  PROC DrawPart48()
    MoveL Offs(pOrigin,340.15,243.37,0.00),v40,z0,tPen\WObj:=wPaper;
    MoveL Offs(pOrigin,341.95,245.18,0.00),v40,z0,tPen\WObj:=wPaper;
    MoveL Offs(pOrigin,341.67,245.49,0.00),v40,z0,tPen\WObj:=wPaper;
    MoveL Offs(pOrigin,344.68,242.48,0.00),v40,z0,tPen\WObj:=wPaper;
    MoveL Offs(pOrigin,344.35,243.09,0.00),v40,z0,tPen\WObj:=wPaper;
    MoveL Offs(pOrigin,346.00,244.74,0.00),v40,z0,tPen\WObj:=wPaper;
    MoveL Offs(pOrigin,346.47,245.17,0.00),v40,z0,tPen\WObj:=wPaper;
    MoveL Offs(pOrigin,349.92,241.72,0.00),v40,z0,tPen\WObj:=wPaper;
    MoveL Offs(pOrigin,349.89,242.65,0.00),v40,z0,tPen\WObj:=wPaper;
    MoveL Offs(pOrigin,351.54,244.31,0.00),v40,z0,tPen\WObj:=wPaper;
    MoveL Offs(pOrigin,351.41,244.71,0.00),v40,z0,tPen\WObj:=wPaper;
    MoveL Offs(pOrigin,354.87,241.25,0.00),v40,z0,tPen\WObj:=wPaper;
    MoveL Offs(pOrigin,355.13,241.92,0.00),v40,z0,tPen\WObj:=wPaper;
    MoveL Offs(pOrigin,356.93,243.72,0.00),v40,z0,tPen\WObj:=wPaper;
    MoveL Offs(pOrigin,356.51,244.09,0.00),v40,z0,tPen\WObj:=wPaper;
    MoveL Offs(pOrigin,362.82,237.78,0.00),v40,z0,tPen\WObj:=wPaper;
    MoveL Offs(pOrigin,363.50,238.35,0.00),v40,z0,tPen\WObj:=wPaper;
    MoveL Offs(pOrigin,366.96,241.81,0.00),v40,z0,tPen\WObj:=wPaper;
    MoveL Offs(pOrigin,367.45,242.11,0.00),v40,z0,tPen\WObj:=wPaper;
    MoveL Offs(pOrigin,373.61,235.95,0.00),v40,z0,tPen\WObj:=wPaper;
    MoveL Offs(pOrigin,372.78,235.68,0.00),v40,z0,tPen\WObj:=wPaper;
    MoveL Offs(pOrigin,371.43,234.33,0.00),v40,z0,tPen\WObj:=wPaper;
    MoveL Offs(pOrigin,371.98,234.65,0.00),v40,z0,tPen\WObj:=wPaper;
    MoveL Offs(pOrigin,373.04,234.65,0.00),v40,z0,tPen\WObj:=wPaper;
    MoveL Offs(pOrigin,373.25,234.93,0.00),v40,z0,tPen\WObj:=wPaper;
    MoveL Offs(pOrigin,372.40,235.77,0.00),v40,z0,tPen\WObj:=wPaper;
    MoveL Offs(pOrigin,373.25,234.93,0.00),v40,z0,tPen\WObj:=wPaper;
    MoveL Offs(pOrigin,373.53,234.94,0.00),v40,z0,tPen\WObj:=wPaper;
    MoveL Offs(pOrigin,372.18,233.58,0.00),v40,z0,tPen\WObj:=wPaper;
    MoveL Offs(pOrigin,372.19,233.65,0.00),v40,z0,tPen\WObj:=wPaper;
    MoveL Offs(pOrigin,371.98,234.07,0.00),v40,z0,tPen\WObj:=wPaper;
    MoveL Offs(pOrigin,372.19,233.65,0.00),v40,z0,tPen\WObj:=wPaper;
    MoveL Offs(pOrigin,372.61,233.44,0.00),v40,z0,tPen\WObj:=wPaper;
    MoveL Offs(pOrigin,372.83,233.01,0.00),v40,z0,tPen\WObj:=wPaper;
    MoveL Offs(pOrigin,372.61,233.44,0.00),v40,z0,tPen\WObj:=wPaper;
    MoveL Offs(pOrigin,372.83,233.59,0.00),v40,z0,tPen\WObj:=wPaper;
    MoveL Offs(pOrigin,373.89,233.59,0.00),v40,z0,tPen\WObj:=wPaper;
    MoveL Offs(pOrigin,374.10,233.86,0.00),v40,z0,tPen\WObj:=wPaper;
    MoveL Offs(pOrigin,373.46,234.50,0.00),v40,z0,tPen\WObj:=wPaper;
    MoveL Offs(pOrigin,374.10,233.86,0.00),v40,z0,tPen\WObj:=wPaper;
    MoveL Offs(pOrigin,374.13,234.04,0.00),v40,z0,tPen\WObj:=wPaper;
    MoveL Offs(pOrigin,372.77,232.69,0.00),v40,z0,tPen\WObj:=wPaper;
    MoveL Offs(pOrigin,373.46,232.54,0.00),v40,z0,tPen\WObj:=wPaper;
    MoveL Offs(pOrigin,374.52,232.54,0.00),v40,z0,tPen\WObj:=wPaper;
    MoveL Offs(pOrigin,374.74,232.80,0.00),v40,z0,tPen\WObj:=wPaper;
    MoveL Offs(pOrigin,374.31,233.44,0.00),v40,z0,tPen\WObj:=wPaper;
    MoveL Offs(pOrigin,374.74,232.80,0.00),v40,z0,tPen\WObj:=wPaper;
    MoveL Offs(pOrigin,374.72,233.14,0.00),v40,z0,tPen\WObj:=wPaper;
    MoveL Offs(pOrigin,373.37,231.79,0.00),v40,z0,tPen\WObj:=wPaper;
    MoveL Offs(pOrigin,373.46,231.95,0.00),v40,z0,tPen\WObj:=wPaper;
    MoveL Offs(pOrigin,373.25,232.38,0.00),v40,z0,tPen\WObj:=wPaper;
    MoveL Offs(pOrigin,373.46,231.95,0.00),v40,z0,tPen\WObj:=wPaper;
    MoveL Offs(pOrigin,373.97,230.89,0.00),v40,z0,tPen\WObj:=wPaper;
    MoveL Offs(pOrigin,375.32,232.25,0.00),v40,z0,tPen\WObj:=wPaper;
    MoveL Offs(pOrigin,375.16,231.95,0.00),v40,z0,tPen\WObj:=wPaper;
    MoveL Offs(pOrigin,374.95,232.38,0.00),v40,z0,tPen\WObj:=wPaper;
    MoveL Offs(pOrigin,375.16,231.95,0.00),v40,z0,tPen\WObj:=wPaper;
    MoveL Offs(pOrigin,375.77,231.20,0.00),v40,z0,tPen\WObj:=wPaper;
    MoveL Offs(pOrigin,374.56,230.00,0.00),v40,z0,tPen\WObj:=wPaper;
    MoveL Offs(pOrigin,373.78,229.81,0.00),v40,z0,tPen\WObj:=wPaper;
    MoveL Offs(pOrigin,377.99,225.60,0.00),v40,z0,tPen\WObj:=wPaper;
    MoveL Offs(pOrigin,377.25,225.21,0.00),v40,z0,tPen\WObj:=wPaper;
    MoveL Offs(pOrigin,375.74,223.71,0.00),v40,fine,tPen\WObj:=wPaper;
    MoveL Offs(pOrigin,375.74,223.71,6.00),v60,z5,tPen\WObj:=wPaper;
    MoveL Offs(pOrigin,375.60,225.06,6.00),vTravel,z5,tPen\WObj:=wPaper;
    MoveL Offs(pOrigin,375.60,225.06,0.00),v60,z0,tPen\WObj:=wPaper;
    MoveL Offs(pOrigin,377.10,226.56,0.00),v40,z0,tPen\WObj:=wPaper;
    MoveL Offs(pOrigin,377.68,227.40,0.00),v40,z0,tPen\WObj:=wPaper;
    MoveL Offs(pOrigin,361.60,243.48,0.00),v40,z0,tPen\WObj:=wPaper;
    MoveL Offs(pOrigin,362.02,242.84,0.00),v40,z0,tPen\WObj:=wPaper;
    MoveL Offs(pOrigin,360.37,241.19,0.00),v40,z0,tPen\WObj:=wPaper;
    MoveL Offs(pOrigin,361.41,240.74,0.00),v40,z0,tPen\WObj:=wPaper;
    MoveL Offs(pOrigin,363.37,242.70,0.00),v40,z0,tPen\WObj:=wPaper;
    MoveL Offs(pOrigin,363.55,243.02,0.00),v40,z0,tPen\WObj:=wPaper;
    MoveL Offs(pOrigin,377.07,229.50,0.00),v40,z0,tPen\WObj:=wPaper;
    MoveL Offs(pOrigin,376.51,228.95,0.00),v40,z0,tPen\WObj:=wPaper;
    MoveL Offs(pOrigin,375.16,227.60,0.00),v40,z0,tPen\WObj:=wPaper;
    MoveL Offs(pOrigin,374.53,227.56,0.00),v40,z0,tPen\WObj:=wPaper;
    MoveL Offs(pOrigin,378.14,223.95,0.00),v40,z0,tPen\WObj:=wPaper;
    MoveL Offs(pOrigin,377.54,224.01,0.00),v40,z0,tPen\WObj:=wPaper;
    MoveL Offs(pOrigin,375.89,222.36,0.00),v40,fine,tPen\WObj:=wPaper;
    MoveL Offs(pOrigin,375.89,222.36,6.00),v60,z5,tPen\WObj:=wPaper;
    MoveL Offs(pOrigin,375.73,220.71,6.00),vTravel,z5,tPen\WObj:=wPaper;
    MoveL Offs(pOrigin,375.73,220.71,0.00),v60,z0,tPen\WObj:=wPaper;
    MoveL Offs(pOrigin,377.69,222.67,0.00),v40,z0,tPen\WObj:=wPaper;
    MoveL Offs(pOrigin,378.29,222.30,0.00),v40,z0,tPen\WObj:=wPaper;
    MoveL Offs(pOrigin,374.84,225.76,0.00),v40,z0,tPen\WObj:=wPaper;
    MoveL Offs(pOrigin,375.30,226.25,0.00),v40,z0,tPen\WObj:=wPaper;
    MoveL Offs(pOrigin,376.80,227.76,0.00),v40,fine,tPen\WObj:=wPaper;
    MoveL Offs(pOrigin,376.80,227.76,6.00),v60,z5,tPen\WObj:=wPaper;
    MoveL Offs(pOrigin,378.13,228.45,6.00),vTravel,z5,tPen\WObj:=wPaper;
    MoveL Offs(pOrigin,378.13,228.45,0.00),v60,z0,tPen\WObj:=wPaper;
    MoveL Offs(pOrigin,385.94,220.63,0.00),v40,z0,tPen\WObj:=wPaper;
    MoveL Offs(pOrigin,385.47,219.99,0.00),v40,z0,tPen\WObj:=wPaper;
    MoveL Offs(pOrigin,383.97,218.49,0.00),v40,fine,tPen\WObj:=wPaper;
    MoveL Offs(pOrigin,383.97,218.49,6.00),v60,z5,tPen\WObj:=wPaper;
    MoveL Offs(pOrigin,383.67,219.69,6.00),vTravel,z5,tPen\WObj:=wPaper;
    MoveL Offs(pOrigin,383.67,219.69,0.00),v60,z0,tPen\WObj:=wPaper;
    MoveL Offs(pOrigin,385.32,221.34,0.00),v40,fine,tPen\WObj:=wPaper;
    MoveL Offs(pOrigin,385.32,221.34,6.00),v60,z5,tPen\WObj:=wPaper;
    MoveL Offs(pOrigin,385.48,222.58,6.00),vTravel,z5,tPen\WObj:=wPaper;
    MoveL Offs(pOrigin,385.48,222.58,0.00),v60,z0,tPen\WObj:=wPaper;
    MoveL Offs(pOrigin,377.37,230.70,0.00),v40,z0,tPen\WObj:=wPaper;
    MoveL Offs(pOrigin,378.31,230.76,0.00),v40,z0,tPen\WObj:=wPaper;
    MoveL Offs(pOrigin,380.87,233.31,0.00),v40,z0,tPen\WObj:=wPaper;
    MoveL Offs(pOrigin,380.69,233.23,0.00),v40,z0,tPen\WObj:=wPaper;
    MoveL Offs(pOrigin,380.26,233.86,0.00),v40,z0,tPen\WObj:=wPaper;
    MoveL Offs(pOrigin,380.69,233.23,0.00),v40,z0,tPen\WObj:=wPaper;
    MoveL Offs(pOrigin,380.69,232.54,0.00),v40,z0,tPen\WObj:=wPaper;
    MoveL Offs(pOrigin,378.56,232.54,0.00),v40,z0,tPen\WObj:=wPaper;
    MoveL Offs(pOrigin,377.87,231.80,0.00),v40,z0,tPen\WObj:=wPaper;
    MoveL Offs(pOrigin,380.12,234.06,0.00),v40,z0,tPen\WObj:=wPaper;
    MoveL Offs(pOrigin,379.84,234.29,0.00),v40,z0,tPen\WObj:=wPaper;
    MoveL Offs(pOrigin,379.41,234.93,0.00),v40,z0,tPen\WObj:=wPaper;
    MoveL Offs(pOrigin,379.84,234.29,0.00),v40,z0,tPen\WObj:=wPaper;
    MoveL Offs(pOrigin,380.05,233.59,0.00),v40,z0,tPen\WObj:=wPaper;
    MoveL Offs(pOrigin,377.71,233.59,0.00),v40,z0,tPen\WObj:=wPaper;
    MoveL Offs(pOrigin,377.50,233.44,0.00),v40,z0,tPen\WObj:=wPaper;
    MoveL Offs(pOrigin,377.50,232.59,0.00),v40,z0,tPen\WObj:=wPaper;
    MoveL Offs(pOrigin,378.99,228.55,0.00),v40,z0,tPen\WObj:=wPaper;
  ENDPROC

  PROC DrawPart49()
    MoveL Offs(pOrigin,379.62,225.79,0.00),v40,z0,tPen\WObj:=wPaper;
    MoveL Offs(pOrigin,380.48,217.93,0.00),v40,z0,tPen\WObj:=wPaper;
    MoveL Offs(pOrigin,380.26,204.75,0.00),v40,z0,tPen\WObj:=wPaper;
    MoveL Offs(pOrigin,378.35,186.90,0.00),v40,z0,tPen\WObj:=wPaper;
    MoveL Offs(pOrigin,378.35,186.90,0.00),v40,z0,tPen\WObj:=wPaper;
    MoveL Offs(pOrigin,377.92,185.84,0.00),v40,z0,tPen\WObj:=wPaper;
    MoveL Offs(pOrigin,378.77,185.62,0.00),v40,z0,tPen\WObj:=wPaper;
    MoveL Offs(pOrigin,378.77,185.62,0.00),v40,z0,tPen\WObj:=wPaper;
    MoveL Offs(pOrigin,378.56,182.65,0.00),v40,z0,tPen\WObj:=wPaper;
    MoveL Offs(pOrigin,379.20,179.25,0.00),v40,z0,tPen\WObj:=wPaper;
    MoveL Offs(pOrigin,381.75,171.39,0.00),v40,z0,tPen\WObj:=wPaper;
    MoveL Offs(pOrigin,381.75,169.26,0.00),v40,z0,tPen\WObj:=wPaper;
    MoveL Offs(pOrigin,380.90,166.93,0.00),v40,z0,tPen\WObj:=wPaper;
    MoveL Offs(pOrigin,380.90,164.80,0.00),v40,z0,tPen\WObj:=wPaper;
    MoveL Offs(pOrigin,382.53,159.91,0.00),v40,z0,tPen\WObj:=wPaper;
    MoveL Offs(pOrigin,385.01,155.02,0.00),v40,z0,tPen\WObj:=wPaper;
    MoveL Offs(pOrigin,387.06,149.71,0.00),v40,z0,tPen\WObj:=wPaper;
    MoveL Offs(pOrigin,387.27,147.16,0.00),v40,z0,tPen\WObj:=wPaper;
    MoveL Offs(pOrigin,386.85,144.61,0.00),v40,z0,tPen\WObj:=wPaper;
    MoveL Offs(pOrigin,387.13,143.76,0.00),v40,z0,tPen\WObj:=wPaper;
    MoveL Offs(pOrigin,389.54,141.43,0.00),v40,z0,tPen\WObj:=wPaper;
    MoveL Offs(pOrigin,390.46,139.30,0.00),v40,z0,tPen\WObj:=wPaper;
    MoveL Offs(pOrigin,391.10,129.95,0.00),v40,z0,tPen\WObj:=wPaper;
    MoveL Offs(pOrigin,391.60,128.68,0.00),v40,z0,tPen\WObj:=wPaper;
    MoveL Offs(pOrigin,392.59,128.46,0.00),v40,z0,tPen\WObj:=wPaper;
    MoveL Offs(pOrigin,392.80,129.31,0.00),v40,z0,tPen\WObj:=wPaper;
    MoveL Offs(pOrigin,388.55,169.69,0.00),v40,z0,tPen\WObj:=wPaper;
    MoveL Offs(pOrigin,384.30,217.50,0.00),v40,z0,tPen\WObj:=wPaper;
    MoveL Offs(pOrigin,383.45,222.39,0.00),v40,z0,tPen\WObj:=wPaper;
    MoveL Offs(pOrigin,381.61,228.55,0.00),v40,z0,tPen\WObj:=wPaper;
    MoveL Offs(pOrigin,380.33,231.10,0.00),v40,z0,tPen\WObj:=wPaper;
    MoveL Offs(pOrigin,379.41,231.52,0.00),v40,z0,tPen\WObj:=wPaper;
    MoveL Offs(pOrigin,379.41,231.52,0.00),v40,z0,tPen\WObj:=wPaper;
    MoveL Offs(pOrigin,378.35,233.30,0.00),v40,z0,tPen\WObj:=wPaper;
    MoveL Offs(pOrigin,377.50,233.44,0.00),v40,z0,tPen\WObj:=wPaper;
    MoveL Offs(pOrigin,377.50,233.44,0.00),v40,z0,tPen\WObj:=wPaper;
    MoveL Offs(pOrigin,377.08,234.50,0.00),v40,z0,tPen\WObj:=wPaper;
    MoveL Offs(pOrigin,375.66,235.42,0.00),v40,z0,tPen\WObj:=wPaper;
    MoveL Offs(pOrigin,373.46,237.69,0.00),v40,z0,tPen\WObj:=wPaper;
    MoveL Offs(pOrigin,373.46,237.82,0.00),v40,z0,tPen\WObj:=wPaper;
    MoveL Offs(pOrigin,375.59,237.82,0.00),v40,z0,tPen\WObj:=wPaper;
    MoveL Offs(pOrigin,375.64,238.54,0.00),v40,z0,tPen\WObj:=wPaper;
    MoveL Offs(pOrigin,373.99,236.89,0.00),v40,z0,tPen\WObj:=wPaper;
    MoveL Offs(pOrigin,374.52,236.84,0.00),v40,z0,tPen\WObj:=wPaper;
    MoveL Offs(pOrigin,374.74,236.41,0.00),v40,z0,tPen\WObj:=wPaper;
    MoveL Offs(pOrigin,374.52,236.84,0.00),v40,z0,tPen\WObj:=wPaper;
    MoveL Offs(pOrigin,374.74,236.76,0.00),v40,z0,tPen\WObj:=wPaper;
    MoveL Offs(pOrigin,377.08,236.76,0.00),v40,z0,tPen\WObj:=wPaper;
    MoveL Offs(pOrigin,377.28,237.20,0.00),v40,z0,tPen\WObj:=wPaper;
    MoveL Offs(pOrigin,375.48,235.39,0.00),v40,z0,tPen\WObj:=wPaper;
    MoveL Offs(pOrigin,375.80,235.70,0.00),v40,z0,tPen\WObj:=wPaper;
    MoveL Offs(pOrigin,378.14,235.70,0.00),v40,z0,tPen\WObj:=wPaper;
    MoveL Offs(pOrigin,378.78,235.70,0.00),v40,z0,tPen\WObj:=wPaper;
    MoveL Offs(pOrigin,376.82,233.75,0.00),v40,z0,tPen\WObj:=wPaper;
    MoveL Offs(pOrigin,376.65,234.65,0.00),v40,z0,tPen\WObj:=wPaper;
    MoveL Offs(pOrigin,379.20,234.65,0.00),v40,z0,tPen\WObj:=wPaper;
    MoveL Offs(pOrigin,379.52,234.96,0.00),v40,z0,tPen\WObj:=wPaper;
    MoveL Offs(pOrigin,377.27,232.70,0.00),v40,fine,tPen\WObj:=wPaper;
    MoveL Offs(pOrigin,377.27,232.70,6.00),v60,z5,tPen\WObj:=wPaper;
    MoveL Offs(pOrigin,376.17,231.90,6.00),vTravel,z5,tPen\WObj:=wPaper;
    MoveL Offs(pOrigin,376.17,231.90,0.00),v60,z0,tPen\WObj:=wPaper;
    MoveL Offs(pOrigin,365.50,242.57,0.00),v40,z0,tPen\WObj:=wPaper;
    MoveL Offs(pOrigin,365.76,242.10,0.00),v40,z0,tPen\WObj:=wPaper;
    MoveL Offs(pOrigin,362.46,238.80,0.00),v40,fine,tPen\WObj:=wPaper;
    MoveL Offs(pOrigin,362.46,238.80,6.00),v60,z5,tPen\WObj:=wPaper;
    MoveL Offs(pOrigin,361.26,239.09,6.00),vTravel,z5,tPen\WObj:=wPaper;
    MoveL Offs(pOrigin,361.26,239.09,0.00),v60,z0,tPen\WObj:=wPaper;
    MoveL Offs(pOrigin,364.72,242.55,0.00),v40,fine,tPen\WObj:=wPaper;
    MoveL Offs(pOrigin,364.72,242.55,6.00),v60,z5,tPen\WObj:=wPaper;
    MoveL Offs(pOrigin,363.26,242.04,6.00),vTravel,z5,tPen\WObj:=wPaper;
    MoveL Offs(pOrigin,363.26,242.04,0.00),v60,z0,tPen\WObj:=wPaper;
    MoveL Offs(pOrigin,356.46,242.04,0.00),v40,z0,tPen\WObj:=wPaper;
    MoveL Offs(pOrigin,356.47,241.78,0.00),v40,z0,tPen\WObj:=wPaper;
    MoveL Offs(pOrigin,358.28,243.58,0.00),v40,z0,tPen\WObj:=wPaper;
    MoveL Offs(pOrigin,358.31,243.79,0.00),v40,z0,tPen\WObj:=wPaper;
    MoveL Offs(pOrigin,364.92,237.18,0.00),v40,z0,tPen\WObj:=wPaper;
    MoveL Offs(pOrigin,364.55,237.91,0.00),v40,z0,tPen\WObj:=wPaper;
    MoveL Offs(pOrigin,368.16,241.51,0.00),v40,z0,tPen\WObj:=wPaper;
    MoveL Offs(pOrigin,367.72,240.98,0.00),v40,z0,tPen\WObj:=wPaper;
    MoveL Offs(pOrigin,362.84,240.98,0.00),v40,fine,tPen\WObj:=wPaper;
    MoveL Offs(pOrigin,362.84,240.98,6.00),v60,z5,tPen\WObj:=wPaper;
    MoveL Offs(pOrigin,361.14,239.39,6.00),vTravel,z5,tPen\WObj:=wPaper;
    MoveL Offs(pOrigin,361.14,239.39,0.00),v60,z0,tPen\WObj:=wPaper;
    MoveL Offs(pOrigin,361.56,238.82,0.00),v40,z0,tPen\WObj:=wPaper;
    MoveL Offs(pOrigin,364.75,238.11,0.00),v40,z0,tPen\WObj:=wPaper;
    MoveL Offs(pOrigin,368.15,236.84,0.00),v40,z0,tPen\WObj:=wPaper;
    MoveL Offs(pOrigin,367.84,236.72,0.00),v40,z0,tPen\WObj:=wPaper;
    MoveL Offs(pOrigin,371.45,240.32,0.00),v40,z0,tPen\WObj:=wPaper;
    MoveL Offs(pOrigin,371.34,239.93,0.00),v40,z0,tPen\WObj:=wPaper;
    MoveL Offs(pOrigin,367.72,239.93,0.00),v40,fine,tPen\WObj:=wPaper;
    MoveL Offs(pOrigin,367.72,239.93,6.00),v60,z5,tPen\WObj:=wPaper;
    MoveL Offs(pOrigin,369.36,241.22,6.00),vTravel,z5,tPen\WObj:=wPaper;
    MoveL Offs(pOrigin,369.36,241.22,0.00),v60,z0,tPen\WObj:=wPaper;
    MoveL Offs(pOrigin,365.90,237.76,0.00),v40,z0,tPen\WObj:=wPaper;
    MoveL Offs(pOrigin,366.66,237.82,0.00),v40,z0,tPen\WObj:=wPaper;
    MoveL Offs(pOrigin,368.58,237.82,0.00),v40,z0,tPen\WObj:=wPaper;
    MoveL Offs(pOrigin,368.79,236.76,0.00),v40,z0,tPen\WObj:=wPaper;
    MoveL Offs(pOrigin,370.49,236.76,0.00),v40,z0,tPen\WObj:=wPaper;
    MoveL Offs(pOrigin,371.14,237.03,0.00),v40,z0,tPen\WObj:=wPaper;
    MoveL Offs(pOrigin,369.79,235.67,0.00),v40,z0,tPen\WObj:=wPaper;
    MoveL Offs(pOrigin,369.85,235.99,0.00),v40,z0,tPen\WObj:=wPaper;
    MoveL Offs(pOrigin,370.27,235.56,0.00),v40,z0,tPen\WObj:=wPaper;
    MoveL Offs(pOrigin,369.85,235.99,0.00),v40,z0,tPen\WObj:=wPaper;
    MoveL Offs(pOrigin,370.49,235.70,0.00),v40,z0,tPen\WObj:=wPaper;
    MoveL Offs(pOrigin,371.76,235.70,0.00),v40,z0,tPen\WObj:=wPaper;
    MoveL Offs(pOrigin,371.76,236.20,0.00),v40,z0,tPen\WObj:=wPaper;
    MoveL Offs(pOrigin,371.34,236.62,0.00),v40,z0,tPen\WObj:=wPaper;
    MoveL Offs(pOrigin,371.76,236.20,0.00),v40,z0,tPen\WObj:=wPaper;
    MoveL Offs(pOrigin,372.04,236.43,0.00),v40,z0,tPen\WObj:=wPaper;
    MoveL Offs(pOrigin,370.69,235.08,0.00),v40,z0,tPen\WObj:=wPaper;
    MoveL Offs(pOrigin,370.70,235.35,0.00),v40,z0,tPen\WObj:=wPaper;
    MoveL Offs(pOrigin,371.12,235.14,0.00),v40,z0,tPen\WObj:=wPaper;
    MoveL Offs(pOrigin,370.70,235.35,0.00),v40,fine,tPen\WObj:=wPaper;
    MoveL Offs(pOrigin,370.70,235.35,6.00),v60,z5,tPen\WObj:=wPaper;
    MoveL Offs(pOrigin,369.00,236.41,6.00),vTravel,z5,tPen\WObj:=wPaper;
    MoveL Offs(pOrigin,369.00,236.41,0.00),v60,z0,tPen\WObj:=wPaper;
    MoveL Offs(pOrigin,369.42,236.20,0.00),v40,z0,tPen\WObj:=wPaper;
    MoveL Offs(pOrigin,369.00,236.41,0.00),v40,z0,tPen\WObj:=wPaper;
    MoveL Offs(pOrigin,368.89,236.27,0.00),v40,z0,tPen\WObj:=wPaper;
    MoveL Offs(pOrigin,372.65,240.03,0.00),v40,z0,tPen\WObj:=wPaper;
  ENDPROC

  PROC DrawPart50()
    MoveL Offs(pOrigin,373.69,239.58,0.00),v40,z0,tPen\WObj:=wPaper;
    MoveL Offs(pOrigin,372.19,238.08,0.00),v40,z0,tPen\WObj:=wPaper;
    MoveL Offs(pOrigin,373.04,237.90,0.00),v40,z0,tPen\WObj:=wPaper;
    MoveL Offs(pOrigin,369.42,239.39,0.00),v40,z0,tPen\WObj:=wPaper;
    MoveL Offs(pOrigin,364.54,240.66,0.00),v40,z0,tPen\WObj:=wPaper;
    MoveL Offs(pOrigin,356.89,241.94,0.00),v40,z0,tPen\WObj:=wPaper;
    MoveL Offs(pOrigin,341.38,243.64,0.00),v40,z0,tPen\WObj:=wPaper;
    MoveL Offs(pOrigin,320.55,244.91,0.00),v40,z0,tPen\WObj:=wPaper;
    MoveL Offs(pOrigin,302.06,245.12,0.00),v40,z0,tPen\WObj:=wPaper;
    MoveL Offs(pOrigin,299.30,244.91,0.00),v40,z0,tPen\WObj:=wPaper;
    MoveL Offs(pOrigin,298.88,244.27,0.00),v40,z0,tPen\WObj:=wPaper;
    MoveL Offs(pOrigin,297.88,240.24,0.00),v40,z0,tPen\WObj:=wPaper;
    MoveL Offs(pOrigin,298.02,239.81,0.00),v40,z0,tPen\WObj:=wPaper;
    MoveL Offs(pOrigin,298.02,239.81,0.00),v40,z0,tPen\WObj:=wPaper;
    MoveL Offs(pOrigin,295.26,237.83,0.00),v40,z0,tPen\WObj:=wPaper;
    MoveL Offs(pOrigin,294.20,237.48,0.00),v40,z0,tPen\WObj:=wPaper;
    MoveL Offs(pOrigin,291.93,237.69,0.00),v40,z0,tPen\WObj:=wPaper;
    MoveL Offs(pOrigin,291.44,233.44,0.00),v40,z0,tPen\WObj:=wPaper;
    MoveL Offs(pOrigin,289.24,226.43,0.00),v40,z0,tPen\WObj:=wPaper;
    MoveL Offs(pOrigin,295.97,218.35,0.00),v40,z0,tPen\WObj:=wPaper;
    MoveL Offs(pOrigin,300.79,213.75,0.00),v40,z0,tPen\WObj:=wPaper;
    MoveL Offs(pOrigin,310.14,211.34,0.00),v40,z0,tPen\WObj:=wPaper;
    MoveL Offs(pOrigin,317.58,208.86,0.00),v40,z0,tPen\WObj:=wPaper;
    MoveL Offs(pOrigin,336.27,201.07,0.00),v40,z0,tPen\WObj:=wPaper;
    MoveL Offs(pOrigin,346.90,197.52,0.00),v40,z0,tPen\WObj:=wPaper;
    MoveL Offs(pOrigin,366.88,192.21,0.00),v40,z0,tPen\WObj:=wPaper;
    MoveL Offs(pOrigin,371.76,190.51,0.00),v40,z0,tPen\WObj:=wPaper;
    MoveL Offs(pOrigin,372.33,190.58,0.00),v40,z0,tPen\WObj:=wPaper;
    MoveL Offs(pOrigin,373.89,196.89,0.00),v40,z0,tPen\WObj:=wPaper;
    MoveL Offs(pOrigin,375.38,205.18,0.00),v40,z0,tPen\WObj:=wPaper;
    MoveL Offs(pOrigin,375.80,208.79,0.00),v40,z0,tPen\WObj:=wPaper;
    MoveL Offs(pOrigin,375.80,216.86,0.00),v40,z0,tPen\WObj:=wPaper;
    MoveL Offs(pOrigin,375.80,216.86,0.00),v40,z0,tPen\WObj:=wPaper;
    MoveL Offs(pOrigin,376.44,217.50,0.00),v40,z0,tPen\WObj:=wPaper;
    MoveL Offs(pOrigin,376.23,218.35,0.00),v40,z0,tPen\WObj:=wPaper;
    MoveL Offs(pOrigin,375.38,218.35,0.00),v40,z0,tPen\WObj:=wPaper;
    MoveL Offs(pOrigin,375.38,217.07,0.00),v40,z0,tPen\WObj:=wPaper;
    MoveL Offs(pOrigin,375.80,216.86,0.00),v40,z0,tPen\WObj:=wPaper;
    MoveL Offs(pOrigin,376.22,216.70,0.00),v40,z0,tPen\WObj:=wPaper;
    MoveL Offs(pOrigin,377.29,216.70,0.00),v40,z0,tPen\WObj:=wPaper;
    MoveL Offs(pOrigin,377.97,216.97,0.00),v40,z0,tPen\WObj:=wPaper;
    MoveL Offs(pOrigin,375.57,214.57,0.00),v40,z0,tPen\WObj:=wPaper;
    MoveL Offs(pOrigin,376.22,214.58,0.00),v40,z0,tPen\WObj:=wPaper;
    MoveL Offs(pOrigin,377.29,214.58,0.00),v40,z0,tPen\WObj:=wPaper;
    MoveL Offs(pOrigin,377.66,213.68,0.00),v40,z0,tPen\WObj:=wPaper;
    MoveL Offs(pOrigin,375.56,211.57,0.00),v40,z0,tPen\WObj:=wPaper;
    MoveL Offs(pOrigin,376.01,211.42,0.00),v40,z0,tPen\WObj:=wPaper;
    MoveL Offs(pOrigin,377.29,211.42,0.00),v40,z0,tPen\WObj:=wPaper;
    MoveL Offs(pOrigin,377.65,210.68,0.00),v40,z0,tPen\WObj:=wPaper;
    MoveL Offs(pOrigin,375.55,208.58,0.00),v40,z0,tPen\WObj:=wPaper;
    MoveL Offs(pOrigin,376.01,209.30,0.00),v40,z0,tPen\WObj:=wPaper;
    MoveL Offs(pOrigin,377.08,209.30,0.00),v40,z0,tPen\WObj:=wPaper;
    MoveL Offs(pOrigin,377.50,209.03,0.00),v40,z0,tPen\WObj:=wPaper;
    MoveL Offs(pOrigin,375.24,206.78,0.00),v40,z0,tPen\WObj:=wPaper;
    MoveL Offs(pOrigin,374.60,206.59,0.00),v40,z0,tPen\WObj:=wPaper;
    MoveL Offs(pOrigin,377.15,204.03,0.00),v40,z0,tPen\WObj:=wPaper;
    MoveL Offs(pOrigin,376.58,203.64,0.00),v40,z0,tPen\WObj:=wPaper;
    MoveL Offs(pOrigin,374.48,201.53,0.00),v40,z0,tPen\WObj:=wPaper;
    MoveL Offs(pOrigin,373.87,201.35,0.00),v40,z0,tPen\WObj:=wPaper;
    MoveL Offs(pOrigin,376.42,198.79,0.00),v40,z0,tPen\WObj:=wPaper;
    MoveL Offs(pOrigin,375.67,198.24,0.00),v40,z0,tPen\WObj:=wPaper;
    MoveL Offs(pOrigin,373.26,195.84,0.00),v40,z0,tPen\WObj:=wPaper;
    MoveL Offs(pOrigin,372.98,196.26,0.00),v40,z0,tPen\WObj:=wPaper;
    MoveL Offs(pOrigin,375.39,193.85,0.00),v40,z0,tPen\WObj:=wPaper;
    MoveL Offs(pOrigin,374.90,194.50,0.00),v40,z0,tPen\WObj:=wPaper;
    MoveL Offs(pOrigin,368.59,188.18,0.00),v40,z0,tPen\WObj:=wPaper;
    MoveL Offs(pOrigin,368.58,187.75,0.00),v40,z0,tPen\WObj:=wPaper;
    MoveL Offs(pOrigin,369.00,188.18,0.00),v40,z0,tPen\WObj:=wPaper;
    MoveL Offs(pOrigin,368.58,187.75,0.00),v40,z0,tPen\WObj:=wPaper;
    MoveL Offs(pOrigin,367.91,187.88,0.00),v40,z0,tPen\WObj:=wPaper;
    MoveL Offs(pOrigin,369.87,185.93,0.00),v40,z0,tPen\WObj:=wPaper;
    MoveL Offs(pOrigin,369.42,186.48,0.00),v40,z0,tPen\WObj:=wPaper;
    MoveL Offs(pOrigin,369.64,186.90,0.00),v40,z0,tPen\WObj:=wPaper;
    MoveL Offs(pOrigin,369.42,186.48,0.00),v40,z0,tPen\WObj:=wPaper;
    MoveL Offs(pOrigin,370.46,186.83,0.00),v40,z0,tPen\WObj:=wPaper;
    MoveL Offs(pOrigin,363.40,193.89,0.00),v40,z0,tPen\WObj:=wPaper;
    MoveL Offs(pOrigin,363.37,193.41,0.00),v40,z0,tPen\WObj:=wPaper;
    MoveL Offs(pOrigin,361.86,191.91,0.00),v40,z0,tPen\WObj:=wPaper;
    MoveL Offs(pOrigin,361.78,192.41,0.00),v40,z0,tPen\WObj:=wPaper;
    MoveL Offs(pOrigin,364.54,192.41,0.00),v40,z0,tPen\WObj:=wPaper;
    MoveL Offs(pOrigin,364.41,192.97,0.00),v40,z0,tPen\WObj:=wPaper;
    MoveL Offs(pOrigin,363.06,191.61,0.00),v40,z0,tPen\WObj:=wPaper;
    MoveL Offs(pOrigin,363.41,190.89,0.00),v40,z0,tPen\WObj:=wPaper;
    MoveL Offs(pOrigin,359.35,194.95,0.00),v40,z0,tPen\WObj:=wPaper;
    MoveL Offs(pOrigin,359.62,194.15,0.00),v40,z0,tPen\WObj:=wPaper;
    MoveL Offs(pOrigin,358.42,192.95,0.00),v40,z0,tPen\WObj:=wPaper;
    MoveL Offs(pOrigin,357.74,193.46,0.00),v40,z0,tPen\WObj:=wPaper;
    MoveL Offs(pOrigin,360.50,193.46,0.00),v40,z0,tPen\WObj:=wPaper;
    MoveL Offs(pOrigin,360.97,194.00,0.00),v40,z0,tPen\WObj:=wPaper;
    MoveL Offs(pOrigin,359.62,192.65,0.00),v40,z0,tPen\WObj:=wPaper;
    MoveL Offs(pOrigin,359.36,191.95,0.00),v40,z0,tPen\WObj:=wPaper;
    MoveL Offs(pOrigin,355.31,196.01,0.00),v40,z0,tPen\WObj:=wPaper;
    MoveL Offs(pOrigin,354.98,195.48,0.00),v40,z0,tPen\WObj:=wPaper;
    MoveL Offs(pOrigin,353.63,194.13,0.00),v40,z0,tPen\WObj:=wPaper;
    MoveL Offs(pOrigin,353.70,194.52,0.00),v40,z0,tPen\WObj:=wPaper;
    MoveL Offs(pOrigin,356.67,194.52,0.00),v40,z0,tPen\WObj:=wPaper;
    MoveL Offs(pOrigin,357.38,194.89,0.00),v40,z0,tPen\WObj:=wPaper;
    MoveL Offs(pOrigin,356.03,193.54,0.00),v40,z0,tPen\WObj:=wPaper;
    MoveL Offs(pOrigin,355.32,193.01,0.00),v40,z0,tPen\WObj:=wPaper;
    MoveL Offs(pOrigin,350.96,197.37,0.00),v40,z0,tPen\WObj:=wPaper;
    MoveL Offs(pOrigin,350.34,196.82,0.00),v40,z0,tPen\WObj:=wPaper;
    MoveL Offs(pOrigin,348.99,195.46,0.00),v40,z0,tPen\WObj:=wPaper;
    MoveL Offs(pOrigin,349.17,194.68,0.00),v40,z0,tPen\WObj:=wPaper;
    MoveL Offs(pOrigin,344.81,199.04,0.00),v40,z0,tPen\WObj:=wPaper;
    MoveL Offs(pOrigin,344.66,198.60,0.00),v40,z0,tPen\WObj:=wPaper;
    MoveL Offs(pOrigin,343.16,197.09,0.00),v40,z0,tPen\WObj:=wPaper;
    MoveL Offs(pOrigin,343.02,196.35,0.00),v40,z0,tPen\WObj:=wPaper;
    MoveL Offs(pOrigin,338.36,201.01,0.00),v40,z0,tPen\WObj:=wPaper;
    MoveL Offs(pOrigin,337.92,200.82,0.00),v40,z0,tPen\WObj:=wPaper;
    MoveL Offs(pOrigin,336.42,199.32,0.00),v40,z0,tPen\WObj:=wPaper;
    MoveL Offs(pOrigin,336.06,199.80,0.00),v40,z0,tPen\WObj:=wPaper;
    MoveL Offs(pOrigin,339.04,199.80,0.00),v40,z0,tPen\WObj:=wPaper;
    MoveL Offs(pOrigin,338.97,200.38,0.00),v40,z0,tPen\WObj:=wPaper;
    MoveL Offs(pOrigin,337.47,198.87,0.00),v40,z0,tPen\WObj:=wPaper;
    MoveL Offs(pOrigin,336.72,198.16,0.00),v40,z0,tPen\WObj:=wPaper;
    MoveL Offs(pOrigin,330.86,204.02,0.00),v40,z0,tPen\WObj:=wPaper;
    MoveL Offs(pOrigin,330.44,203.80,0.00),v40,z0,tPen\WObj:=wPaper;
    MoveL Offs(pOrigin,328.94,202.29,0.00),v40,z0,tPen\WObj:=wPaper;
    MoveL Offs(pOrigin,328.93,201.48,0.00),v40,z0,tPen\WObj:=wPaper;
    MoveL Offs(pOrigin,322.91,207.49,0.00),v40,z0,tPen\WObj:=wPaper;
  ENDPROC

  PROC DrawPart51()
    MoveL Offs(pOrigin,323.11,206.92,0.00),v40,z0,tPen\WObj:=wPaper;
    MoveL Offs(pOrigin,321.61,205.42,0.00),v40,z0,tPen\WObj:=wPaper;
    MoveL Offs(pOrigin,321.13,204.80,0.00),v40,z0,tPen\WObj:=wPaper;
    MoveL Offs(pOrigin,315.72,210.21,0.00),v40,z0,tPen\WObj:=wPaper;
    MoveL Offs(pOrigin,315.63,209.89,0.00),v40,z0,tPen\WObj:=wPaper;
    MoveL Offs(pOrigin,314.13,208.39,0.00),v40,z0,tPen\WObj:=wPaper;
    MoveL Offs(pOrigin,313.78,207.67,0.00),v40,z0,tPen\WObj:=wPaper;
    MoveL Offs(pOrigin,309.12,212.33,0.00),v40,z0,tPen\WObj:=wPaper;
    MoveL Offs(pOrigin,308.75,211.97,0.00),v40,z0,tPen\WObj:=wPaper;
    MoveL Offs(pOrigin,307.09,210.32,0.00),v40,z0,tPen\WObj:=wPaper;
    MoveL Offs(pOrigin,307.48,209.49,0.00),v40,z0,tPen\WObj:=wPaper;
    MoveL Offs(pOrigin,303.12,213.85,0.00),v40,z0,tPen\WObj:=wPaper;
    MoveL Offs(pOrigin,302.91,213.60,0.00),v40,z0,tPen\WObj:=wPaper;
    MoveL Offs(pOrigin,300.66,211.34,0.00),v40,z0,tPen\WObj:=wPaper;
    MoveL Offs(pOrigin,300.79,211.55,0.00),v40,z0,tPen\WObj:=wPaper;
    MoveL Offs(pOrigin,299.30,213.04,0.00),v40,z0,tPen\WObj:=wPaper;
    MoveL Offs(pOrigin,300.79,211.55,0.00),v40,z0,tPen\WObj:=wPaper;
    MoveL Offs(pOrigin,301.00,211.42,0.00),v40,z0,tPen\WObj:=wPaper;
    MoveL Offs(pOrigin,308.65,211.42,0.00),v40,z0,tPen\WObj:=wPaper;
    MoveL Offs(pOrigin,308.44,210.36,0.00),v40,z0,tPen\WObj:=wPaper;
    MoveL Offs(pOrigin,312.05,210.36,0.00),v40,z0,tPen\WObj:=wPaper;
    MoveL Offs(pOrigin,312.19,210.93,0.00),v40,z0,tPen\WObj:=wPaper;
    MoveL Offs(pOrigin,310.69,209.43,0.00),v40,z0,tPen\WObj:=wPaper;
    MoveL Offs(pOrigin,311.73,208.98,0.00),v40,z0,tPen\WObj:=wPaper;
    MoveL Offs(pOrigin,313.24,210.48,0.00),v40,z0,tPen\WObj:=wPaper;
    MoveL Offs(pOrigin,313.32,211.12,0.00),v40,z0,tPen\WObj:=wPaper;
    MoveL Offs(pOrigin,318.58,205.86,0.00),v40,z0,tPen\WObj:=wPaper;
    MoveL Offs(pOrigin,318.47,206.76,0.00),v40,z0,tPen\WObj:=wPaper;
    MoveL Offs(pOrigin,319.97,208.26,0.00),v40,z0,tPen\WObj:=wPaper;
    MoveL Offs(pOrigin,320.36,208.55,0.00),v40,z0,tPen\WObj:=wPaper;
    MoveL Offs(pOrigin,326.23,202.69,0.00),v40,z0,tPen\WObj:=wPaper;
    MoveL Offs(pOrigin,326.85,203.19,0.00),v40,z0,tPen\WObj:=wPaper;
    MoveL Offs(pOrigin,328.35,204.69,0.00),v40,z0,tPen\WObj:=wPaper;
    MoveL Offs(pOrigin,328.16,205.23,0.00),v40,z0,tPen\WObj:=wPaper;
    MoveL Offs(pOrigin,334.18,199.22,0.00),v40,z0,tPen\WObj:=wPaper;
    MoveL Offs(pOrigin,334.33,200.21,0.00),v40,z0,tPen\WObj:=wPaper;
    MoveL Offs(pOrigin,335.83,201.72,0.00),v40,z0,tPen\WObj:=wPaper;
    MoveL Offs(pOrigin,335.81,202.06,0.00),v40,z0,tPen\WObj:=wPaper;
    MoveL Offs(pOrigin,340.92,196.95,0.00),v40,z0,tPen\WObj:=wPaper;
    MoveL Offs(pOrigin,340.91,197.84,0.00),v40,z0,tPen\WObj:=wPaper;
    MoveL Offs(pOrigin,342.41,199.34,0.00),v40,z0,tPen\WObj:=wPaper;
    MoveL Offs(pOrigin,342.86,199.49,0.00),v40,z0,tPen\WObj:=wPaper;
    MoveL Offs(pOrigin,347.37,194.99,0.00),v40,z0,tPen\WObj:=wPaper;
    MoveL Offs(pOrigin,347.64,195.61,0.00),v40,z0,tPen\WObj:=wPaper;
    MoveL Offs(pOrigin,349.15,197.11,0.00),v40,z0,tPen\WObj:=wPaper;
    MoveL Offs(pOrigin,349.02,196.63,0.00),v40,z0,tPen\WObj:=wPaper;
    MoveL Offs(pOrigin,346.26,196.63,0.00),v40,z0,tPen\WObj:=wPaper;
    MoveL Offs(pOrigin,346.60,196.06,0.00),v40,z0,tPen\WObj:=wPaper;
    MoveL Offs(pOrigin,347.95,197.41,0.00),v40,z0,tPen\WObj:=wPaper;
    MoveL Offs(pOrigin,346.90,197.85,0.00),v40,z0,tPen\WObj:=wPaper;
    MoveL Offs(pOrigin,345.55,196.50,0.00),v40,z0,tPen\WObj:=wPaper;
    MoveL Offs(pOrigin,345.27,195.59,0.00),v40,z0,tPen\WObj:=wPaper;
    MoveL Offs(pOrigin,340.46,200.40,0.00),v40,z0,tPen\WObj:=wPaper;
    MoveL Offs(pOrigin,340.17,200.08,0.00),v40,z0,tPen\WObj:=wPaper;
    MoveL Offs(pOrigin,338.67,198.58,0.00),v40,z0,tPen\WObj:=wPaper;
    MoveL Offs(pOrigin,339.25,198.74,0.00),v40,z0,tPen\WObj:=wPaper;
    MoveL Offs(pOrigin,342.22,198.74,0.00),v40,z0,tPen\WObj:=wPaper;
    MoveL Offs(pOrigin,342.44,197.69,0.00),v40,z0,tPen\WObj:=wPaper;
    MoveL Offs(pOrigin,345.41,197.69,0.00),v40,z0,tPen\WObj:=wPaper;
    MoveL Offs(pOrigin,345.71,198.15,0.00),v40,z0,tPen\WObj:=wPaper;
    MoveL Offs(pOrigin,344.20,196.65,0.00),v40,fine,tPen\WObj:=wPaper;
    MoveL Offs(pOrigin,344.20,196.65,6.00),v60,z5,tPen\WObj:=wPaper;
    MoveL Offs(pOrigin,341.96,197.39,6.00),vTravel,z5,tPen\WObj:=wPaper;
    MoveL Offs(pOrigin,341.96,197.39,0.00),v60,z0,tPen\WObj:=wPaper;
    MoveL Offs(pOrigin,343.46,198.89,0.00),v40,fine,tPen\WObj:=wPaper;
    MoveL Offs(pOrigin,343.46,198.89,6.00),v60,z5,tPen\WObj:=wPaper;
    MoveL Offs(pOrigin,341.22,199.63,6.00),vTravel,z5,tPen\WObj:=wPaper;
    MoveL Offs(pOrigin,341.22,199.63,0.00),v60,z0,tPen\WObj:=wPaper;
    MoveL Offs(pOrigin,339.86,198.28,0.00),v40,fine,tPen\WObj:=wPaper;
    MoveL Offs(pOrigin,339.86,198.28,6.00),v60,z5,tPen\WObj:=wPaper;
    MoveL Offs(pOrigin,338.82,197.56,6.00),vTravel,z5,tPen\WObj:=wPaper;
    MoveL Offs(pOrigin,338.82,197.56,0.00),v60,z0,tPen\WObj:=wPaper;
    MoveL Offs(pOrigin,333.41,202.97,0.00),v40,z0,tPen\WObj:=wPaper;
    MoveL Offs(pOrigin,333.73,202.61,0.00),v40,z0,tPen\WObj:=wPaper;
    MoveL Offs(pOrigin,332.08,200.96,0.00),v40,z0,tPen\WObj:=wPaper;
    MoveL Offs(pOrigin,331.63,200.28,0.00),v40,z0,tPen\WObj:=wPaper;
    MoveL Offs(pOrigin,325.46,206.44,0.00),v40,z0,tPen\WObj:=wPaper;
    MoveL Offs(pOrigin,325.21,206.03,0.00),v40,z0,tPen\WObj:=wPaper;
    MoveL Offs(pOrigin,323.70,204.52,0.00),v40,z0,tPen\WObj:=wPaper;
    MoveL Offs(pOrigin,323.52,205.08,0.00),v40,z0,tPen\WObj:=wPaper;
    MoveL Offs(pOrigin,326.08,205.08,0.00),v40,z0,tPen\WObj:=wPaper;
    MoveL Offs(pOrigin,326.25,205.58,0.00),v40,z0,tPen\WObj:=wPaper;
    MoveL Offs(pOrigin,324.90,204.23,0.00),v40,z0,tPen\WObj:=wPaper;
    MoveL Offs(pOrigin,325.86,204.02,0.00),v40,z0,tPen\WObj:=wPaper;
    MoveL Offs(pOrigin,328.41,204.02,0.00),v40,z0,tPen\WObj:=wPaper;
    MoveL Offs(pOrigin,327.77,204.75,0.00),v40,z0,tPen\WObj:=wPaper;
    MoveL Offs(pOrigin,328.20,204.54,0.00),v40,z0,tPen\WObj:=wPaper;
    MoveL Offs(pOrigin,327.77,204.75,0.00),v40,z0,tPen\WObj:=wPaper;
    MoveL Offs(pOrigin,327.30,205.13,0.00),v40,z0,tPen\WObj:=wPaper;
    MoveL Offs(pOrigin,325.95,203.78,0.00),v40,fine,tPen\WObj:=wPaper;
    MoveL Offs(pOrigin,325.95,203.78,6.00),v60,z5,tPen\WObj:=wPaper;
    MoveL Offs(pOrigin,327.89,202.74,6.00),vTravel,z5,tPen\WObj:=wPaper;
    MoveL Offs(pOrigin,327.89,202.74,0.00),v60,z0,tPen\WObj:=wPaper;
    MoveL Offs(pOrigin,329.40,204.24,0.00),v40,fine,tPen\WObj:=wPaper;
    MoveL Offs(pOrigin,329.40,204.24,6.00),v60,z5,tPen\WObj:=wPaper;
    MoveL Offs(pOrigin,328.41,202.97,6.00),vTravel,z5,tPen\WObj:=wPaper;
    MoveL Offs(pOrigin,328.41,202.97,0.00),v60,z0,tPen\WObj:=wPaper;
    MoveL Offs(pOrigin,330.96,202.97,0.00),v40,z0,tPen\WObj:=wPaper;
    MoveL Offs(pOrigin,331.49,203.35,0.00),v40,z0,tPen\WObj:=wPaper;
    MoveL Offs(pOrigin,329.99,201.85,0.00),v40,z0,tPen\WObj:=wPaper;
    MoveL Offs(pOrigin,330.75,201.91,0.00),v40,z0,tPen\WObj:=wPaper;
    MoveL Offs(pOrigin,333.51,201.91,0.00),v40,z0,tPen\WObj:=wPaper;
    MoveL Offs(pOrigin,333.30,200.86,0.00),v40,z0,tPen\WObj:=wPaper;
    MoveL Offs(pOrigin,336.06,200.86,0.00),v40,z0,tPen\WObj:=wPaper;
    MoveL Offs(pOrigin,336.88,201.27,0.00),v40,z0,tPen\WObj:=wPaper;
    MoveL Offs(pOrigin,335.37,199.77,0.00),v40,fine,tPen\WObj:=wPaper;
    MoveL Offs(pOrigin,335.37,199.77,6.00),v60,z5,tPen\WObj:=wPaper;
    MoveL Offs(pOrigin,334.63,202.01,6.00),vTravel,z5,tPen\WObj:=wPaper;
    MoveL Offs(pOrigin,334.63,202.01,0.00),v60,z0,tPen\WObj:=wPaper;
    MoveL Offs(pOrigin,333.13,200.51,0.00),v40,fine,tPen\WObj:=wPaper;
    MoveL Offs(pOrigin,333.13,200.51,6.00),v60,z5,tPen\WObj:=wPaper;
    MoveL Offs(pOrigin,331.03,201.40,6.00),vTravel,z5,tPen\WObj:=wPaper;
    MoveL Offs(pOrigin,331.03,201.40,0.00),v60,z0,tPen\WObj:=wPaper;
    MoveL Offs(pOrigin,332.54,202.90,0.00),v40,fine,tPen\WObj:=wPaper;
    MoveL Offs(pOrigin,332.54,202.90,6.00),v60,z5,tPen\WObj:=wPaper;
    MoveL Offs(pOrigin,331.63,198.78,6.00),vTravel,z5,tPen\WObj:=wPaper;
    MoveL Offs(pOrigin,331.63,198.78,0.00),v60,z0,tPen\WObj:=wPaper;
    MoveL Offs(pOrigin,333.73,196.68,0.00),v40,fine,tPen\WObj:=wPaper;
    MoveL Offs(pOrigin,333.73,196.68,6.00),v60,z5,tPen\WObj:=wPaper;
    MoveL Offs(pOrigin,331.78,197.13,6.00),vTravel,z5,tPen\WObj:=wPaper;
  ENDPROC

  PROC DrawPart52()
    MoveL Offs(pOrigin,331.78,197.13,0.00),v60,z0,tPen\WObj:=wPaper;
    MoveL Offs(pOrigin,329.08,199.84,0.00),v40,fine,tPen\WObj:=wPaper;
    MoveL Offs(pOrigin,329.08,199.84,6.00),v60,z5,tPen\WObj:=wPaper;
    MoveL Offs(pOrigin,327.44,198.49,6.00),vTravel,z5,tPen\WObj:=wPaper;
    MoveL Offs(pOrigin,327.44,198.49,0.00),v60,z0,tPen\WObj:=wPaper;
    MoveL Offs(pOrigin,324.28,201.65,0.00),v40,fine,tPen\WObj:=wPaper;
    MoveL Offs(pOrigin,324.28,201.65,6.00),v60,z5,tPen\WObj:=wPaper;
    MoveL Offs(pOrigin,322.25,201.35,6.00),vTravel,z5,tPen\WObj:=wPaper;
    MoveL Offs(pOrigin,322.25,201.35,0.00),v60,z0,tPen\WObj:=wPaper;
    MoveL Offs(pOrigin,321.83,201.92,0.00),v40,z0,tPen\WObj:=wPaper;
    MoveL Offs(pOrigin,317.79,203.26,0.00),v40,z0,tPen\WObj:=wPaper;
    MoveL Offs(pOrigin,312.69,204.54,0.00),v40,z0,tPen\WObj:=wPaper;
    MoveL Offs(pOrigin,308.01,205.25,0.00),v40,z0,tPen\WObj:=wPaper;
    MoveL Offs(pOrigin,303.83,210.27,0.00),v40,z0,tPen\WObj:=wPaper;
    MoveL Offs(pOrigin,303.41,211.48,0.00),v40,z0,tPen\WObj:=wPaper;
    MoveL Offs(pOrigin,309.50,210.06,0.00),v40,z0,tPen\WObj:=wPaper;
    MoveL Offs(pOrigin,317.58,207.37,0.00),v40,z0,tPen\WObj:=wPaper;
    MoveL Offs(pOrigin,333.94,200.43,0.00),v40,z0,tPen\WObj:=wPaper;
    MoveL Offs(pOrigin,342.86,197.31,0.00),v40,z0,tPen\WObj:=wPaper;
    MoveL Offs(pOrigin,365.60,191.15,0.00),v40,z0,tPen\WObj:=wPaper;
    MoveL Offs(pOrigin,369.64,189.80,0.00),v40,z0,tPen\WObj:=wPaper;
    MoveL Offs(pOrigin,369.85,189.45,0.00),v40,z0,tPen\WObj:=wPaper;
    MoveL Offs(pOrigin,366.95,184.56,0.00),v40,z0,tPen\WObj:=wPaper;
    MoveL Offs(pOrigin,365.53,181.16,0.00),v40,z0,tPen\WObj:=wPaper;
    MoveL Offs(pOrigin,360.50,165.23,0.00),v40,z0,tPen\WObj:=wPaper;
    MoveL Offs(pOrigin,353.91,139.30,0.00),v40,z0,tPen\WObj:=wPaper;
    MoveL Offs(pOrigin,348.17,111.68,0.00),v40,z0,tPen\WObj:=wPaper;
    MoveL Offs(pOrigin,344.42,99.99,0.00),v40,z0,tPen\WObj:=wPaper;
    MoveL Offs(pOrigin,342.01,93.61,0.00),v40,z0,tPen\WObj:=wPaper;
    MoveL Offs(pOrigin,342.23,93.12,0.00),v40,z0,tPen\WObj:=wPaper;
    MoveL Offs(pOrigin,342.79,93.40,0.00),v40,z0,tPen\WObj:=wPaper;
    MoveL Offs(pOrigin,345.55,100.41,0.00),v40,z0,tPen\WObj:=wPaper;
    MoveL Offs(pOrigin,346.33,101.47,0.00),v40,z0,tPen\WObj:=wPaper;
    MoveL Offs(pOrigin,347.54,105.72,0.00),v40,z0,tPen\WObj:=wPaper;
    MoveL Offs(pOrigin,346.48,105.82,0.00),v40,z0,tPen\WObj:=wPaper;
    MoveL Offs(pOrigin,350.51,105.82,0.00),v40,z0,tPen\WObj:=wPaper;
    MoveL Offs(pOrigin,351.11,104.99,0.00),v40,z0,tPen\WObj:=wPaper;
    MoveL Offs(pOrigin,342.55,96.43,0.00),v40,z0,tPen\WObj:=wPaper;
    MoveL Offs(pOrigin,342.28,97.03,0.00),v40,z0,tPen\WObj:=wPaper;
    MoveL Offs(pOrigin,346.49,92.83,0.00),v40,z0,tPen\WObj:=wPaper;
    MoveL Offs(pOrigin,345.83,92.24,0.00),v40,z0,tPen\WObj:=wPaper;
    MoveL Offs(pOrigin,342.52,88.94,0.00),v40,fine,tPen\WObj:=wPaper;
    MoveL Offs(pOrigin,342.52,88.94,6.00),v60,z5,tPen\WObj:=wPaper;
    MoveL Offs(pOrigin,341.18,89.08,6.00),vTravel,z5,tPen\WObj:=wPaper;
    MoveL Offs(pOrigin,341.18,89.08,0.00),v60,z0,tPen\WObj:=wPaper;
    MoveL Offs(pOrigin,338.92,86.83,0.00),v40,z0,tPen\WObj:=wPaper;
    MoveL Offs(pOrigin,338.56,87.31,0.00),v40,z0,tPen\WObj:=wPaper;
    MoveL Offs(pOrigin,342.77,83.10,0.00),v40,z0,tPen\WObj:=wPaper;
    MoveL Offs(pOrigin,343.22,84.15,0.00),v40,z0,tPen\WObj:=wPaper;
    MoveL Offs(pOrigin,338.86,88.51,0.00),v40,z0,tPen\WObj:=wPaper;
    MoveL Offs(pOrigin,339.31,89.55,0.00),v40,z0,tPen\WObj:=wPaper;
    MoveL Offs(pOrigin,343.66,85.19,0.00),v40,z0,tPen\WObj:=wPaper;
    MoveL Offs(pOrigin,343.11,85.04,0.00),v40,z0,tPen\WObj:=wPaper;
    MoveL Offs(pOrigin,339.96,81.89,0.00),v40,fine,tPen\WObj:=wPaper;
    MoveL Offs(pOrigin,339.96,81.89,6.00),v60,z5,tPen\WObj:=wPaper;
    MoveL Offs(pOrigin,341.75,82.19,6.00),vTravel,z5,tPen\WObj:=wPaper;
    MoveL Offs(pOrigin,341.75,82.19,0.00),v60,z0,tPen\WObj:=wPaper;
    MoveL Offs(pOrigin,338.90,79.34,0.00),v40,z0,tPen\WObj:=wPaper;
    MoveL Offs(pOrigin,338.59,79.82,0.00),v40,z0,tPen\WObj:=wPaper;
    MoveL Offs(pOrigin,340.39,78.01,0.00),v40,z0,tPen\WObj:=wPaper;
    MoveL Offs(pOrigin,340.84,79.06,0.00),v40,z0,tPen\WObj:=wPaper;
    MoveL Offs(pOrigin,336.78,83.12,0.00),v40,z0,tPen\WObj:=wPaper;
    MoveL Offs(pOrigin,336.33,82.07,0.00),v40,z0,tPen\WObj:=wPaper;
    MoveL Offs(pOrigin,337.83,80.57,0.00),v40,z0,tPen\WObj:=wPaper;
    MoveL Offs(pOrigin,337.24,79.67,0.00),v40,z0,tPen\WObj:=wPaper;
    MoveL Offs(pOrigin,336.04,80.87,0.00),v40,z0,tPen\WObj:=wPaper;
    MoveL Offs(pOrigin,335.59,79.83,0.00),v40,z0,tPen\WObj:=wPaper;
    MoveL Offs(pOrigin,336.64,78.78,0.00),v40,z0,tPen\WObj:=wPaper;
    MoveL Offs(pOrigin,336.20,77.73,0.00),v40,z0,tPen\WObj:=wPaper;
    MoveL Offs(pOrigin,335.14,78.78,0.00),v40,z0,tPen\WObj:=wPaper;
    MoveL Offs(pOrigin,334.70,77.73,0.00),v40,z0,tPen\WObj:=wPaper;
    MoveL Offs(pOrigin,339.66,72.77,0.00),v40,z0,tPen\WObj:=wPaper;
    MoveL Offs(pOrigin,339.46,72.79,0.00),v40,z0,tPen\WObj:=wPaper;
    MoveL Offs(pOrigin,342.44,72.79,0.00),v40,z0,tPen\WObj:=wPaper;
    MoveL Offs(pOrigin,347.33,72.15,0.00),v40,z0,tPen\WObj:=wPaper;
    MoveL Offs(pOrigin,353.06,70.88,0.00),v40,z0,tPen\WObj:=wPaper;
    MoveL Offs(pOrigin,358.80,69.03,0.00),v40,z0,tPen\WObj:=wPaper;
    MoveL Offs(pOrigin,363.05,67.33,0.00),v40,z0,tPen\WObj:=wPaper;
    MoveL Offs(pOrigin,368.79,64.36,0.00),v40,z0,tPen\WObj:=wPaper;
    MoveL Offs(pOrigin,373.25,61.53,0.00),v40,z0,tPen\WObj:=wPaper;
    MoveL Offs(pOrigin,376.65,58.76,0.00),v40,z0,tPen\WObj:=wPaper;
    MoveL Offs(pOrigin,377.08,58.55,0.00),v40,z0,tPen\WObj:=wPaper;
    MoveL Offs(pOrigin,384.73,50.90,0.00),v40,fine,tPen\WObj:=wPaper;
    MoveL Offs(pOrigin,384.73,50.90,6.00),v60,z5,tPen\WObj:=wPaper;
    MoveL Offs(pOrigin,382.39,48.14,6.00),vTravel,z5,tPen\WObj:=wPaper;
    MoveL Offs(pOrigin,382.39,48.14,0.00),v60,z0,tPen\WObj:=wPaper;
    MoveL Offs(pOrigin,381.75,48.78,0.00),v40,z0,tPen\WObj:=wPaper;
    MoveL Offs(pOrigin,382.39,48.14,0.00),v40,fine,tPen\WObj:=wPaper;
    MoveL Offs(pOrigin,382.39,48.14,6.00),v60,z5,tPen\WObj:=wPaper;
    MoveL Offs(pOrigin,384.09,46.44,6.00),vTravel,z5,tPen\WObj:=wPaper;
    MoveL Offs(pOrigin,384.09,46.44,0.00),v60,z0,tPen\WObj:=wPaper;
    MoveL Offs(pOrigin,382.60,47.92,0.00),v40,z0,tPen\WObj:=wPaper;
    MoveL Offs(pOrigin,384.09,46.44,0.00),v40,fine,tPen\WObj:=wPaper;
    MoveL Offs(pOrigin,384.09,46.44,6.00),v60,z5,tPen\WObj:=wPaper;
    MoveL Offs(pOrigin,386.18,44.17,6.00),vTravel,z5,tPen\WObj:=wPaper;
    MoveL Offs(pOrigin,386.18,44.17,0.00),v60,z0,tPen\WObj:=wPaper;
    MoveL Offs(pOrigin,373.41,56.94,0.00),v40,fine,tPen\WObj:=wPaper;
    MoveL Offs(pOrigin,373.41,56.94,6.00),v60,z5,tPen\WObj:=wPaper;
    MoveL Offs(pOrigin,371.91,56.95,6.00),vTravel,z5,tPen\WObj:=wPaper;
    MoveL Offs(pOrigin,371.91,56.95,0.00),v60,z0,tPen\WObj:=wPaper;
    MoveL Offs(pOrigin,378.37,50.48,0.00),v40,z0,tPen\WObj:=wPaper;
    MoveL Offs(pOrigin,379.20,51.11,0.00),v40,z0,tPen\WObj:=wPaper;
    MoveL Offs(pOrigin,377.71,52.60,0.00),v40,z0,tPen\WObj:=wPaper;
    MoveL Offs(pOrigin,379.20,51.11,0.00),v40,fine,tPen\WObj:=wPaper;
    MoveL Offs(pOrigin,379.20,51.11,6.00),v60,z5,tPen\WObj:=wPaper;
    MoveL Offs(pOrigin,380.91,53.92,6.00),vTravel,z5,tPen\WObj:=wPaper;
    MoveL Offs(pOrigin,380.91,53.92,0.00),v60,z0,tPen\WObj:=wPaper;
    MoveL Offs(pOrigin,369.94,64.89,0.00),v40,z0,tPen\WObj:=wPaper;
    MoveL Offs(pOrigin,370.01,64.16,0.00),v40,z0,tPen\WObj:=wPaper;
    MoveL Offs(pOrigin,369.26,63.40,0.00),v40,z0,tPen\WObj:=wPaper;
    MoveL Offs(pOrigin,368.36,64.00,0.00),v40,z0,tPen\WObj:=wPaper;
    MoveL Offs(pOrigin,369.11,64.75,0.00),v40,z0,tPen\WObj:=wPaper;
    MoveL Offs(pOrigin,368.22,65.35,0.00),v40,z0,tPen\WObj:=wPaper;
    MoveL Offs(pOrigin,367.32,64.45,0.00),v40,z0,tPen\WObj:=wPaper;
    MoveL Offs(pOrigin,366.42,65.04,0.00),v40,z0,tPen\WObj:=wPaper;
    MoveL Offs(pOrigin,367.17,65.79,0.00),v40,z0,tPen\WObj:=wPaper;
    MoveL Offs(pOrigin,366.64,66.70,0.00),v40,z0,tPen\WObj:=wPaper;
    MoveL Offs(pOrigin,374.15,59.19,0.00),v40,fine,tPen\WObj:=wPaper;
    MoveL Offs(pOrigin,374.15,59.19,6.00),v60,z5,tPen\WObj:=wPaper;
    MoveL Offs(pOrigin,374.89,61.43,6.00),vTravel,z5,tPen\WObj:=wPaper;
  ENDPROC

  PROC DrawPart53()
    MoveL Offs(pOrigin,374.89,61.43,0.00),v60,z0,tPen\WObj:=wPaper;
    MoveL Offs(pOrigin,381.66,54.67,0.00),v40,fine,tPen\WObj:=wPaper;
    MoveL Offs(pOrigin,381.66,54.67,6.00),v60,z5,tPen\WObj:=wPaper;
    MoveL Offs(pOrigin,369.42,59.61,6.00),vTravel,z5,tPen\WObj:=wPaper;
    MoveL Offs(pOrigin,369.42,59.61,0.00),v60,z0,tPen\WObj:=wPaper;
    MoveL Offs(pOrigin,377.92,52.60,0.00),v40,z0,tPen\WObj:=wPaper;
    MoveL Offs(pOrigin,387.91,42.61,0.00),v40,fine,tPen\WObj:=wPaper;
    MoveL Offs(pOrigin,387.91,42.61,6.00),v60,z5,tPen\WObj:=wPaper;
    MoveL Offs(pOrigin,386.00,39.00,6.00),vTravel,z5,tPen\WObj:=wPaper;
    MoveL Offs(pOrigin,386.00,39.00,0.00),v60,z0,tPen\WObj:=wPaper;
    MoveL Offs(pOrigin,377.08,37.02,0.00),v40,z0,tPen\WObj:=wPaper;
    MoveL Offs(pOrigin,376.23,36.31,0.00),v40,z0,tPen\WObj:=wPaper;
    MoveL Offs(pOrigin,368.15,33.40,0.00),v40,z0,tPen\WObj:=wPaper;
    MoveL Offs(pOrigin,367.73,32.84,0.00),v40,z0,tPen\WObj:=wPaper;
    MoveL Offs(pOrigin,367.73,32.84,0.00),v40,z0,tPen\WObj:=wPaper;
    MoveL Offs(pOrigin,368.58,32.62,0.00),v40,z0,tPen\WObj:=wPaper;
    MoveL Offs(pOrigin,382.60,34.54,0.00),v40,z0,tPen\WObj:=wPaper;
    MoveL Offs(pOrigin,394.29,36.66,0.00),v40,z0,tPen\WObj:=wPaper;
    MoveL Offs(pOrigin,400.02,38.15,0.00),v40,z0,tPen\WObj:=wPaper;
    MoveL Offs(pOrigin,406.40,40.70,0.00),v40,z0,tPen\WObj:=wPaper;
    MoveL Offs(pOrigin,407.67,42.33,0.00),v40,z0,tPen\WObj:=wPaper;
    MoveL Offs(pOrigin,408.31,42.61,0.00),v40,z0,tPen\WObj:=wPaper;
    MoveL Offs(pOrigin,408.31,42.61,0.00),v40,z0,tPen\WObj:=wPaper;
    MoveL Offs(pOrigin,409.80,43.04,0.00),v40,z0,tPen\WObj:=wPaper;
    MoveL Offs(pOrigin,412.00,45.80,0.00),v40,z0,tPen\WObj:=wPaper;
    MoveL Offs(pOrigin,413.48,48.99,0.00),v40,z0,tPen\WObj:=wPaper;
    MoveL Offs(pOrigin,414.48,52.39,0.00),v40,z0,tPen\WObj:=wPaper;
    MoveL Offs(pOrigin,414.90,55.15,0.00),v40,z0,tPen\WObj:=wPaper;
    MoveL Offs(pOrigin,414.90,58.76,0.00),v40,z0,tPen\WObj:=wPaper;
    MoveL Offs(pOrigin,414.26,62.80,0.00),v40,z0,tPen\WObj:=wPaper;
    MoveL Offs(pOrigin,413.55,65.14,0.00),v40,z0,tPen\WObj:=wPaper;
    MoveL Offs(pOrigin,411.08,68.75,0.00),v40,z0,tPen\WObj:=wPaper;
    MoveL Offs(pOrigin,408.10,71.72,0.00),v40,z0,tPen\WObj:=wPaper;
    MoveL Offs(pOrigin,404.91,74.28,0.00),v40,z0,tPen\WObj:=wPaper;
    MoveL Offs(pOrigin,400.24,77.32,0.00),v40,z0,tPen\WObj:=wPaper;
    MoveL Offs(pOrigin,394.50,80.30,0.00),v40,z0,tPen\WObj:=wPaper;
    MoveL Offs(pOrigin,387.70,82.78,0.00),v40,z0,tPen\WObj:=wPaper;
    MoveL Offs(pOrigin,381.33,84.05,0.00),v40,z0,tPen\WObj:=wPaper;
    MoveL Offs(pOrigin,376.01,83.84,0.00),v40,z0,tPen\WObj:=wPaper;
    MoveL Offs(pOrigin,368.36,81.15,0.00),v40,z0,tPen\WObj:=wPaper;
    MoveL Offs(pOrigin,367.30,79.94,0.00),v40,z0,tPen\WObj:=wPaper;
    MoveL Offs(pOrigin,365.17,79.30,0.00),v40,z0,tPen\WObj:=wPaper;
    MoveL Offs(pOrigin,362.91,77.68,0.00),v40,z0,tPen\WObj:=wPaper;
    MoveL Offs(pOrigin,363.26,77.25,0.00),v40,z0,tPen\WObj:=wPaper;
    MoveL Offs(pOrigin,368.15,77.04,0.00),v40,z0,tPen\WObj:=wPaper;
    MoveL Offs(pOrigin,368.65,76.61,0.00),v40,z0,tPen\WObj:=wPaper;
    MoveL Offs(pOrigin,368.15,76.19,0.00),v40,z0,tPen\WObj:=wPaper;
    MoveL Offs(pOrigin,360.29,76.40,0.00),v40,z0,tPen\WObj:=wPaper;
    MoveL Offs(pOrigin,356.67,76.19,0.00),v40,z0,tPen\WObj:=wPaper;
    MoveL Offs(pOrigin,337.76,73.85,0.00),v40,z0,tPen\WObj:=wPaper;
    MoveL Offs(pOrigin,327.56,72.15,0.00),v40,z0,tPen\WObj:=wPaper;
    MoveL Offs(pOrigin,319.91,70.45,0.00),v40,z0,tPen\WObj:=wPaper;
    MoveL Offs(pOrigin,316.51,69.32,0.00),v40,z0,tPen\WObj:=wPaper;
    MoveL Offs(pOrigin,316.30,68.75,0.00),v40,z0,tPen\WObj:=wPaper;
    MoveL Offs(pOrigin,316.30,68.75,0.00),v40,z0,tPen\WObj:=wPaper;
    MoveL Offs(pOrigin,322.25,68.54,0.00),v40,z0,tPen\WObj:=wPaper;
    MoveL Offs(pOrigin,326.71,67.19,0.00),v40,z0,tPen\WObj:=wPaper;
    MoveL Offs(pOrigin,330.75,65.21,0.00),v40,z0,tPen\WObj:=wPaper;
    MoveL Offs(pOrigin,335.00,62.38,0.00),v40,z0,tPen\WObj:=wPaper;
    MoveL Offs(pOrigin,337.98,59.83,0.00),v40,z0,tPen\WObj:=wPaper;
    MoveL Offs(pOrigin,343.08,54.09,0.00),v40,z0,tPen\WObj:=wPaper;
    MoveL Offs(pOrigin,347.82,46.65,0.00),v40,z0,tPen\WObj:=wPaper;
    MoveL Offs(pOrigin,349.95,42.19,0.00),v40,z0,tPen\WObj:=wPaper;
    MoveL Offs(pOrigin,350.94,39.00,0.00),v40,z0,tPen\WObj:=wPaper;
    MoveL Offs(pOrigin,350.94,34.54,0.00),v40,z0,tPen\WObj:=wPaper;
    MoveL Offs(pOrigin,350.02,31.56,0.00),v40,z0,tPen\WObj:=wPaper;
    MoveL Offs(pOrigin,347.96,28.16,0.00),v40,z0,tPen\WObj:=wPaper;
    MoveL Offs(pOrigin,346.05,26.46,0.00),v40,z0,tPen\WObj:=wPaper;
    MoveL Offs(pOrigin,346.05,25.90,0.00),v40,z0,tPen\WObj:=wPaper;
    MoveL Offs(pOrigin,347.11,25.83,0.00),v40,z0,tPen\WObj:=wPaper;
    MoveL Offs(pOrigin,350.73,27.03,0.00),v40,z0,tPen\WObj:=wPaper;
    MoveL Offs(pOrigin,360.71,31.70,0.00),v40,z0,tPen\WObj:=wPaper;
    MoveL Offs(pOrigin,367.94,34.61,0.00),v40,z0,tPen\WObj:=wPaper;
    MoveL Offs(pOrigin,376.01,37.09,0.00),v40,z0,tPen\WObj:=wPaper;
    MoveL Offs(pOrigin,376.65,36.88,0.00),v40,z0,tPen\WObj:=wPaper;
    MoveL Offs(pOrigin,376.67,36.46,0.00),v40,z0,tPen\WObj:=wPaper;
    MoveL Offs(pOrigin,377.57,37.36,0.00),v40,z0,tPen\WObj:=wPaper;
    MoveL Offs(pOrigin,377.36,38.05,0.00),v40,z0,tPen\WObj:=wPaper;
    MoveL Offs(pOrigin,379.02,36.40,0.00),v40,z0,tPen\WObj:=wPaper;
    MoveL Offs(pOrigin,377.97,35.96,0.00),v40,z0,tPen\WObj:=wPaper;
    MoveL Offs(pOrigin,376.16,37.76,0.00),v40,z0,tPen\WObj:=wPaper;
    MoveL Offs(pOrigin,375.92,37.21,0.00),v40,z0,tPen\WObj:=wPaper;
    MoveL Offs(pOrigin,374.42,35.71,0.00),v40,fine,tPen\WObj:=wPaper;
    MoveL Offs(pOrigin,374.42,35.71,6.00),v60,z5,tPen\WObj:=wPaper;
    MoveL Offs(pOrigin,374.12,36.90,6.00),vTravel,z5,tPen\WObj:=wPaper;
    MoveL Offs(pOrigin,374.12,36.90,0.00),v60,z0,tPen\WObj:=wPaper;
    MoveL Offs(pOrigin,368.41,31.19,0.00),v40,z0,tPen\WObj:=wPaper;
    MoveL Offs(pOrigin,368.55,30.44,0.00),v40,z0,tPen\WObj:=wPaper;
    MoveL Offs(pOrigin,364.79,34.20,0.00),v40,z0,tPen\WObj:=wPaper;
    MoveL Offs(pOrigin,365.27,34.03,0.00),v40,z0,tPen\WObj:=wPaper;
    MoveL Offs(pOrigin,360.92,29.67,0.00),v40,z0,tPen\WObj:=wPaper;
    MoveL Offs(pOrigin,360.50,29.78,0.00),v40,z0,tPen\WObj:=wPaper;
    MoveL Offs(pOrigin,357.52,29.78,0.00),v40,fine,tPen\WObj:=wPaper;
    MoveL Offs(pOrigin,357.52,29.78,6.00),v60,z5,tPen\WObj:=wPaper;
    MoveL Offs(pOrigin,358.67,28.92,6.00),vTravel,z5,tPen\WObj:=wPaper;
    MoveL Offs(pOrigin,358.67,28.92,0.00),v60,z0,tPen\WObj:=wPaper;
    MoveL Offs(pOrigin,362.72,32.97,0.00),v40,z0,tPen\WObj:=wPaper;
    MoveL Offs(pOrigin,362.70,33.31,0.00),v40,z0,tPen\WObj:=wPaper;
    MoveL Offs(pOrigin,365.85,30.15,0.00),v40,z0,tPen\WObj:=wPaper;
    MoveL Offs(pOrigin,364.81,30.58,0.00),v40,z0,tPen\WObj:=wPaper;
    MoveL Offs(pOrigin,369.77,35.54,0.00),v40,z0,tPen\WObj:=wPaper;
    MoveL Offs(pOrigin,369.13,35.83,0.00),v40,z0,tPen\WObj:=wPaper;
    MoveL Offs(pOrigin,373.94,31.02,0.00),v40,z0,tPen\WObj:=wPaper;
    MoveL Offs(pOrigin,373.21,31.51,0.00),v40,z0,tPen\WObj:=wPaper;
    MoveL Offs(pOrigin,375.61,33.91,0.00),v40,z0,tPen\WObj:=wPaper;
    MoveL Offs(pOrigin,376.47,34.46,0.00),v40,z0,tPen\WObj:=wPaper;
    MoveL Offs(pOrigin,379.18,31.76,0.00),v40,z0,tPen\WObj:=wPaper;
    MoveL Offs(pOrigin,378.30,32.12,0.00),v40,z0,tPen\WObj:=wPaper;
    MoveL Offs(pOrigin,380.71,34.53,0.00),v40,z0,tPen\WObj:=wPaper;
    MoveL Offs(pOrigin,380.90,34.01,0.00),v40,z0,tPen\WObj:=wPaper;
    MoveL Offs(pOrigin,387.28,34.01,0.00),v40,z0,tPen\WObj:=wPaper;
    MoveL Offs(pOrigin,387.29,33.65,0.00),v40,z0,tPen\WObj:=wPaper;
    MoveL Offs(pOrigin,389.70,36.05,0.00),v40,z0,tPen\WObj:=wPaper;
    MoveL Offs(pOrigin,389.50,36.37,0.00),v40,z0,tPen\WObj:=wPaper;
    MoveL Offs(pOrigin,391.91,33.97,0.00),v40,z0,tPen\WObj:=wPaper;
    MoveL Offs(pOrigin,391.04,34.41,0.00),v40,z0,tPen\WObj:=wPaper;
    MoveL Offs(pOrigin,393.60,36.96,0.00),v40,z0,tPen\WObj:=wPaper;
    MoveL Offs(pOrigin,393.09,37.26,0.00),v40,z0,tPen\WObj:=wPaper;
    MoveL Offs(pOrigin,395.65,34.70,0.00),v40,z0,tPen\WObj:=wPaper;
    MoveL Offs(pOrigin,394.79,35.17,0.00),v40,z0,tPen\WObj:=wPaper;
  ENDPROC

  PROC DrawPart54()
    MoveL Offs(pOrigin,397.49,37.87,0.00),v40,z0,tPen\WObj:=wPaper;
    MoveL Offs(pOrigin,396.84,37.99,0.00),v40,z0,tPen\WObj:=wPaper;
    MoveL Offs(pOrigin,399.24,35.59,0.00),v40,z0,tPen\WObj:=wPaper;
    MoveL Offs(pOrigin,398.69,36.08,0.00),v40,z0,tPen\WObj:=wPaper;
    MoveL Offs(pOrigin,401.99,39.39,0.00),v40,z0,tPen\WObj:=wPaper;
    MoveL Offs(pOrigin,402.52,39.78,0.00),v40,z0,tPen\WObj:=wPaper;
    MoveL Offs(pOrigin,404.93,37.37,0.00),v40,z0,tPen\WObj:=wPaper;
    MoveL Offs(pOrigin,405.28,38.20,0.00),v40,z0,tPen\WObj:=wPaper;
    MoveL Offs(pOrigin,415.05,47.97,0.00),v40,z0,tPen\WObj:=wPaper;
    MoveL Offs(pOrigin,415.53,47.67,0.00),v40,z0,tPen\WObj:=wPaper;
    MoveL Offs(pOrigin,412.83,50.38,0.00),v40,z0,tPen\WObj:=wPaper;
    MoveL Offs(pOrigin,413.56,50.96,0.00),v40,z0,tPen\WObj:=wPaper;
    MoveL Offs(pOrigin,416.72,54.11,0.00),v40,z0,tPen\WObj:=wPaper;
    MoveL Offs(pOrigin,416.17,54.07,0.00),v40,z0,tPen\WObj:=wPaper;
    MoveL Offs(pOrigin,414.90,54.07,0.00),v40,z0,tPen\WObj:=wPaper;
    MoveL Offs(pOrigin,414.17,54.55,0.00),v40,z0,tPen\WObj:=wPaper;
    MoveL Offs(pOrigin,417.18,57.56,0.00),v40,z0,tPen\WObj:=wPaper;
    MoveL Offs(pOrigin,417.45,57.71,0.00),v40,z0,tPen\WObj:=wPaper;
    MoveL Offs(pOrigin,413.24,61.91,0.00),v40,z0,tPen\WObj:=wPaper;
    MoveL Offs(pOrigin,414.04,61.89,0.00),v40,z0,tPen\WObj:=wPaper;
    MoveL Offs(pOrigin,416.15,64.00,0.00),v40,z0,tPen\WObj:=wPaper;
    MoveL Offs(pOrigin,415.75,63.58,0.00),v40,z0,tPen\WObj:=wPaper;
    MoveL Offs(pOrigin,414.05,63.58,0.00),v40,z0,tPen\WObj:=wPaper;
    MoveL Offs(pOrigin,413.75,63.09,0.00),v40,z0,tPen\WObj:=wPaper;
    MoveL Offs(pOrigin,416.45,65.80,0.00),v40,z0,tPen\WObj:=wPaper;
    MoveL Offs(pOrigin,416.67,65.95,0.00),v40,z0,tPen\WObj:=wPaper;
    MoveL Offs(pOrigin,397.14,85.48,0.00),v40,z0,tPen\WObj:=wPaper;
    MoveL Offs(pOrigin,397.04,85.21,0.00),v40,z0,tPen\WObj:=wPaper;
    MoveL Offs(pOrigin,395.24,83.41,0.00),v40,z0,tPen\WObj:=wPaper;
    MoveL Offs(pOrigin,395.78,83.64,0.00),v40,z0,tPen\WObj:=wPaper;
    MoveL Offs(pOrigin,398.33,83.64,0.00),v40,z0,tPen\WObj:=wPaper;
    MoveL Offs(pOrigin,398.98,84.17,0.00),v40,z0,tPen\WObj:=wPaper;
    MoveL Offs(pOrigin,397.48,82.66,0.00),v40,z0,tPen\WObj:=wPaper;
    MoveL Offs(pOrigin,398.54,82.58,0.00),v40,z0,tPen\WObj:=wPaper;
    MoveL Offs(pOrigin,400.66,82.58,0.00),v40,z0,tPen\WObj:=wPaper;
    MoveL Offs(pOrigin,400.93,83.12,0.00),v40,z0,tPen\WObj:=wPaper;
    MoveL Offs(pOrigin,399.43,81.62,0.00),v40,z0,tPen\WObj:=wPaper;
    MoveL Offs(pOrigin,400.45,81.53,0.00),v40,z0,tPen\WObj:=wPaper;
    MoveL Offs(pOrigin,402.36,81.53,0.00),v40,z0,tPen\WObj:=wPaper;
    MoveL Offs(pOrigin,402.36,81.71,0.00),v40,z0,tPen\WObj:=wPaper;
    MoveL Offs(pOrigin,402.65,81.57,0.00),v40,z0,tPen\WObj:=wPaper;
    MoveL Offs(pOrigin,398.33,84.12,0.00),v40,z0,tPen\WObj:=wPaper;
    MoveL Offs(pOrigin,393.86,85.75,0.00),v40,z0,tPen\WObj:=wPaper;
    MoveL Offs(pOrigin,389.61,86.60,0.00),v40,z0,tPen\WObj:=wPaper;
    MoveL Offs(pOrigin,384.73,86.81,0.00),v40,z0,tPen\WObj:=wPaper;
    MoveL Offs(pOrigin,377.50,85.75,0.00),v40,z0,tPen\WObj:=wPaper;
    MoveL Offs(pOrigin,371.12,83.91,0.00),v40,z0,tPen\WObj:=wPaper;
    MoveL Offs(pOrigin,366.02,81.57,0.00),v40,z0,tPen\WObj:=wPaper;
    MoveL Offs(pOrigin,360.92,78.45,0.00),v40,z0,tPen\WObj:=wPaper;
    MoveL Offs(pOrigin,359.01,77.68,0.00),v40,z0,tPen\WObj:=wPaper;
    MoveL Offs(pOrigin,356.04,77.46,0.00),v40,z0,tPen\WObj:=wPaper;
    MoveL Offs(pOrigin,355.40,77.89,0.00),v40,z0,tPen\WObj:=wPaper;
    MoveL Offs(pOrigin,355.40,77.89,0.00),v40,z0,tPen\WObj:=wPaper;
    MoveL Offs(pOrigin,354.55,77.46,0.00),v40,z0,tPen\WObj:=wPaper;
    MoveL Offs(pOrigin,354.20,77.68,0.00),v40,z0,tPen\WObj:=wPaper;
    MoveL Offs(pOrigin,353.70,79.80,0.00),v40,z0,tPen\WObj:=wPaper;
    MoveL Offs(pOrigin,353.06,87.88,0.00),v40,z0,tPen\WObj:=wPaper;
    MoveL Offs(pOrigin,353.27,91.28,0.00),v40,z0,tPen\WObj:=wPaper;
    MoveL Offs(pOrigin,353.27,91.28,0.00),v40,z0,tPen\WObj:=wPaper;
    MoveL Offs(pOrigin,353.49,92.12,0.00),v40,z0,tPen\WObj:=wPaper;
    MoveL Offs(pOrigin,353.06,92.34,0.00),v40,z0,tPen\WObj:=wPaper;
    MoveL Offs(pOrigin,353.06,92.34,0.00),v40,z0,tPen\WObj:=wPaper;
    MoveL Offs(pOrigin,354.05,95.74,0.00),v40,z0,tPen\WObj:=wPaper;
    MoveL Offs(pOrigin,355.12,97.86,0.00),v40,z0,tPen\WObj:=wPaper;
    MoveL Offs(pOrigin,357.74,101.47,0.00),v40,fine,tPen\WObj:=wPaper;
    MoveL Offs(pOrigin,357.74,101.47,6.00),v60,z5,tPen\WObj:=wPaper;
    MoveL Offs(pOrigin,355.75,99.99,6.00),vTravel,z5,tPen\WObj:=wPaper;
    MoveL Offs(pOrigin,355.75,99.99,0.00),v60,z0,tPen\WObj:=wPaper;
    MoveL Offs(pOrigin,356.65,99.09,0.00),v40,z0,tPen\WObj:=wPaper;
    MoveL Offs(pOrigin,356.21,98.04,0.00),v40,z0,tPen\WObj:=wPaper;
    MoveL Offs(pOrigin,355.15,99.09,0.00),v40,z0,tPen\WObj:=wPaper;
    MoveL Offs(pOrigin,354.41,98.34,0.00),v40,z0,tPen\WObj:=wPaper;
    MoveL Offs(pOrigin,355.76,96.99,0.00),v40,z0,tPen\WObj:=wPaper;
    MoveL Offs(pOrigin,354.98,96.91,0.00),v40,z0,tPen\WObj:=wPaper;
    MoveL Offs(pOrigin,353.18,95.11,0.00),v40,z0,tPen\WObj:=wPaper;
    MoveL Offs(pOrigin,352.77,95.50,0.00),v40,z0,tPen\WObj:=wPaper;
    MoveL Offs(pOrigin,354.57,93.70,0.00),v40,z0,tPen\WObj:=wPaper;
    MoveL Offs(pOrigin,353.92,92.87,0.00),v40,z0,tPen\WObj:=wPaper;
    MoveL Offs(pOrigin,347.91,86.86,0.00),v40,z0,tPen\WObj:=wPaper;
    MoveL Offs(pOrigin,348.39,86.81,0.00),v40,z0,tPen\WObj:=wPaper;
    MoveL Offs(pOrigin,349.88,86.81,0.00),v40,z0,tPen\WObj:=wPaper;
    MoveL Offs(pOrigin,349.88,85.75,0.00),v40,z0,tPen\WObj:=wPaper;
    MoveL Offs(pOrigin,348.39,85.75,0.00),v40,z0,tPen\WObj:=wPaper;
    MoveL Offs(pOrigin,347.61,85.06,0.00),v40,z0,tPen\WObj:=wPaper;
    MoveL Offs(pOrigin,353.62,91.07,0.00),v40,z0,tPen\WObj:=wPaper;
    MoveL Offs(pOrigin,353.28,91.03,0.00),v40,z0,tPen\WObj:=wPaper;
    MoveL Offs(pOrigin,348.60,91.03,0.00),v40,z0,tPen\WObj:=wPaper;
    MoveL Offs(pOrigin,348.07,91.50,0.00),v40,z0,tPen\WObj:=wPaper;
    MoveL Offs(pOrigin,350.93,94.36,0.00),v40,z0,tPen\WObj:=wPaper;
    MoveL Offs(pOrigin,350.72,94.20,0.00),v40,z0,tPen\WObj:=wPaper;
    MoveL Offs(pOrigin,348.39,94.20,0.00),v40,z0,tPen\WObj:=wPaper;
    MoveL Offs(pOrigin,348.39,94.46,0.00),v40,z0,tPen\WObj:=wPaper;
    MoveL Offs(pOrigin,347.96,95.10,0.00),v40,z0,tPen\WObj:=wPaper;
    MoveL Offs(pOrigin,348.39,94.46,0.00),v40,z0,tPen\WObj:=wPaper;
    MoveL Offs(pOrigin,347.93,94.35,0.00),v40,z0,tPen\WObj:=wPaper;
    MoveL Offs(pOrigin,349.89,96.30,0.00),v40,z0,tPen\WObj:=wPaper;
    MoveL Offs(pOrigin,349.45,96.31,0.00),v40,z0,tPen\WObj:=wPaper;
    MoveL Offs(pOrigin,345.20,96.31,0.00),v40,z0,tPen\WObj:=wPaper;
    MoveL Offs(pOrigin,345.41,97.37,0.00),v40,z0,tPen\WObj:=wPaper;
    MoveL Offs(pOrigin,349.24,97.37,0.00),v40,z0,tPen\WObj:=wPaper;
    MoveL Offs(pOrigin,349.59,97.50,0.00),v40,z0,tPen\WObj:=wPaper;
    MoveL Offs(pOrigin,343.28,91.19,0.00),v40,z0,tPen\WObj:=wPaper;
    MoveL Offs(pOrigin,342.68,92.08,0.00),v40,z0,tPen\WObj:=wPaper;
    MoveL Offs(pOrigin,339.98,89.38,0.00),v40,fine,tPen\WObj:=wPaper;
    MoveL Offs(pOrigin,339.98,89.38,6.00),v60,z5,tPen\WObj:=wPaper;
    MoveL Offs(pOrigin,339.75,90.60,6.00),vTravel,z5,tPen\WObj:=wPaper;
    MoveL Offs(pOrigin,339.75,90.60,0.00),v60,z0,tPen\WObj:=wPaper;
    MoveL Offs(pOrigin,344.11,86.24,0.00),v40,z0,tPen\WObj:=wPaper;
    MoveL Offs(pOrigin,344.56,87.29,0.00),v40,z0,tPen\WObj:=wPaper;
    MoveL Offs(pOrigin,340.20,91.65,0.00),v40,z0,tPen\WObj:=wPaper;
    MoveL Offs(pOrigin,340.88,91.78,0.00),v40,z0,tPen\WObj:=wPaper;
    MoveL Offs(pOrigin,360.42,111.31,0.00),v40,z0,tPen\WObj:=wPaper;
    MoveL Offs(pOrigin,360.36,111.81,0.00),v40,z0,tPen\WObj:=wPaper;
    MoveL Offs(pOrigin,362.31,109.85,0.00),v40,z0,tPen\WObj:=wPaper;
    MoveL Offs(pOrigin,363.21,110.45,0.00),v40,z0,tPen\WObj:=wPaper;
    MoveL Offs(pOrigin,361.41,112.25,0.00),v40,z0,tPen\WObj:=wPaper;
    MoveL Offs(pOrigin,362.30,112.85,0.00),v40,z0,tPen\WObj:=wPaper;
    MoveL Offs(pOrigin,364.11,111.05,0.00),v40,z0,tPen\WObj:=wPaper;
    MoveL Offs(pOrigin,363.11,111.02,0.00),v40,z0,tPen\WObj:=wPaper;
    MoveL Offs(pOrigin,367.02,114.93,0.00),v40,z0,tPen\WObj:=wPaper;
  ENDPROC

  PROC DrawPart55()
    MoveL Offs(pOrigin,367.09,115.53,0.00),v40,z0,tPen\WObj:=wPaper;
    MoveL Offs(pOrigin,368.89,113.73,0.00),v40,z0,tPen\WObj:=wPaper;
    MoveL Offs(pOrigin,369.79,114.33,0.00),v40,z0,tPen\WObj:=wPaper;
    MoveL Offs(pOrigin,368.14,115.98,0.00),v40,z0,tPen\WObj:=wPaper;
    MoveL Offs(pOrigin,369.03,116.57,0.00),v40,z0,tPen\WObj:=wPaper;
    MoveL Offs(pOrigin,370.84,114.77,0.00),v40,z0,tPen\WObj:=wPaper;
    MoveL Offs(pOrigin,370.17,115.09,0.00),v40,z0,tPen\WObj:=wPaper;
    MoveL Offs(pOrigin,373.17,118.09,0.00),v40,z0,tPen\WObj:=wPaper;
    MoveL Offs(pOrigin,373.07,118.51,0.00),v40,z0,tPen\WObj:=wPaper;
    MoveL Offs(pOrigin,374.87,116.71,0.00),v40,z0,tPen\WObj:=wPaper;
    MoveL Offs(pOrigin,373.98,116.11,0.00),v40,z0,tPen\WObj:=wPaper;
    MoveL Offs(pOrigin,372.17,117.91,0.00),v40,z0,tPen\WObj:=wPaper;
    MoveL Offs(pOrigin,371.13,117.47,0.00),v40,z0,tPen\WObj:=wPaper;
    MoveL Offs(pOrigin,372.78,115.81,0.00),v40,z0,tPen\WObj:=wPaper;
    MoveL Offs(pOrigin,372.87,116.29,0.00),v40,z0,tPen\WObj:=wPaper;
    MoveL Offs(pOrigin,376.02,119.45,0.00),v40,z0,tPen\WObj:=wPaper;
    MoveL Offs(pOrigin,376.06,120.00,0.00),v40,z0,tPen\WObj:=wPaper;
    MoveL Offs(pOrigin,377.87,118.20,0.00),v40,z0,tPen\WObj:=wPaper;
    MoveL Offs(pOrigin,378.76,118.79,0.00),v40,z0,tPen\WObj:=wPaper;
    MoveL Offs(pOrigin,377.11,120.44,0.00),v40,z0,tPen\WObj:=wPaper;
    MoveL Offs(pOrigin,378.16,120.89,0.00),v40,z0,tPen\WObj:=wPaper;
    MoveL Offs(pOrigin,379.81,119.24,0.00),v40,z0,tPen\WObj:=wPaper;
    MoveL Offs(pOrigin,379.32,119.76,0.00),v40,z0,tPen\WObj:=wPaper;
    MoveL Offs(pOrigin,381.12,121.56,0.00),v40,z0,tPen\WObj:=wPaper;
    MoveL Offs(pOrigin,381.30,122.23,0.00),v40,z0,tPen\WObj:=wPaper;
    MoveL Offs(pOrigin,382.95,120.58,0.00),v40,z0,tPen\WObj:=wPaper;
    MoveL Offs(pOrigin,382.17,121.12,0.00),v40,z0,tPen\WObj:=wPaper;
    MoveL Offs(pOrigin,383.22,122.17,0.00),v40,z0,tPen\WObj:=wPaper;
    MoveL Offs(pOrigin,383.39,123.12,0.00),v40,z0,tPen\WObj:=wPaper;
    MoveL Offs(pOrigin,384.90,121.62,0.00),v40,z0,tPen\WObj:=wPaper;
    MoveL Offs(pOrigin,385.94,122.07,0.00),v40,z0,tPen\WObj:=wPaper;
    MoveL Offs(pOrigin,384.59,123.42,0.00),v40,fine,tPen\WObj:=wPaper;
    MoveL Offs(pOrigin,384.59,123.42,6.00),v60,z5,tPen\WObj:=wPaper;
    MoveL Offs(pOrigin,384.89,124.62,6.00),vTravel,z5,tPen\WObj:=wPaper;
    MoveL Offs(pOrigin,384.89,124.62,0.00),v60,z0,tPen\WObj:=wPaper;
    MoveL Offs(pOrigin,382.93,126.57,0.00),v40,z0,tPen\WObj:=wPaper;
    MoveL Offs(pOrigin,381.89,126.12,0.00),v40,z0,tPen\WObj:=wPaper;
    MoveL Offs(pOrigin,383.69,124.32,0.00),v40,z0,tPen\WObj:=wPaper;
    MoveL Offs(pOrigin,383.38,125.31,0.00),v40,z0,tPen\WObj:=wPaper;
    MoveL Offs(pOrigin,384.28,126.22,0.00),v40,z0,tPen\WObj:=wPaper;
    MoveL Offs(pOrigin,384.28,126.71,0.00),v40,z0,tPen\WObj:=wPaper;
    MoveL Offs(pOrigin,386.23,124.76,0.00),v40,z0,tPen\WObj:=wPaper;
    MoveL Offs(pOrigin,386.83,125.77,0.00),v40,z0,tPen\WObj:=wPaper;
    MoveL Offs(pOrigin,394.04,132.99,0.00),v40,z0,tPen\WObj:=wPaper;
    MoveL Offs(pOrigin,393.65,133.27,0.00),v40,z0,tPen\WObj:=wPaper;
    MoveL Offs(pOrigin,392.38,133.27,0.00),v40,z0,tPen\WObj:=wPaper;
    MoveL Offs(pOrigin,392.38,134.33,0.00),v40,z0,tPen\WObj:=wPaper;
    MoveL Offs(pOrigin,393.44,134.33,0.00),v40,z0,tPen\WObj:=wPaper;
    MoveL Offs(pOrigin,394.04,134.48,0.00),v40,z0,tPen\WObj:=wPaper;
    MoveL Offs(pOrigin,389.09,129.53,0.00),v40,z0,tPen\WObj:=wPaper;
    MoveL Offs(pOrigin,388.46,130.00,0.00),v40,z0,tPen\WObj:=wPaper;
    MoveL Offs(pOrigin,392.37,126.09,0.00),v40,z0,tPen\WObj:=wPaper;
    MoveL Offs(pOrigin,392.07,126.54,0.00),v40,z0,tPen\WObj:=wPaper;
    MoveL Offs(pOrigin,394.63,129.09,0.00),v40,z0,tPen\WObj:=wPaper;
    MoveL Offs(pOrigin,394.29,129.05,0.00),v40,z0,tPen\WObj:=wPaper;
    MoveL Offs(pOrigin,389.83,129.05,0.00),v40,z0,tPen\WObj:=wPaper;
    MoveL Offs(pOrigin,390.73,129.10,0.00),v40,z0,tPen\WObj:=wPaper;
    MoveL Offs(pOrigin,390.73,127.40,0.00),v40,z0,tPen\WObj:=wPaper;
    MoveL Offs(pOrigin,390.42,126.38,0.00),v40,z0,tPen\WObj:=wPaper;
    MoveL Offs(pOrigin,394.48,130.44,0.00),v40,z0,tPen\WObj:=wPaper;
    MoveL Offs(pOrigin,394.08,130.10,0.00),v40,z0,tPen\WObj:=wPaper;
    MoveL Offs(pOrigin,392.80,130.10,0.00),v40,z0,tPen\WObj:=wPaper;
    MoveL Offs(pOrigin,392.59,131.16,0.00),v40,z0,tPen\WObj:=wPaper;
    MoveL Offs(pOrigin,393.86,131.16,0.00),v40,z0,tPen\WObj:=wPaper;
    MoveL Offs(pOrigin,394.19,131.64,0.00),v40,z0,tPen\WObj:=wPaper;
    MoveL Offs(pOrigin,388.48,125.93,0.00),v40,z0,tPen\WObj:=wPaper;
    MoveL Offs(pOrigin,388.63,125.35,0.00),v40,z0,tPen\WObj:=wPaper;
    MoveL Offs(pOrigin,386.53,127.46,0.00),v40,z0,tPen\WObj:=wPaper;
    MoveL Offs(pOrigin,386.68,127.12,0.00),v40,z0,tPen\WObj:=wPaper;
    MoveL Offs(pOrigin,384.88,125.32,0.00),v40,z0,tPen\WObj:=wPaper;
    MoveL Offs(pOrigin,384.51,125.70,0.00),v40,z0,tPen\WObj:=wPaper;
    MoveL Offs(pOrigin,384.94,126.27,0.00),v40,z0,tPen\WObj:=wPaper;
    MoveL Offs(pOrigin,390.04,127.82,0.00),v40,z0,tPen\WObj:=wPaper;
    MoveL Offs(pOrigin,389.19,132.07,0.00),v40,z0,tPen\WObj:=wPaper;
    MoveL Offs(pOrigin,389.19,136.96,0.00),v40,z0,tPen\WObj:=wPaper;
    MoveL Offs(pOrigin,388.41,140.15,0.00),v40,z0,tPen\WObj:=wPaper;
    MoveL Offs(pOrigin,385.36,143.41,0.00),v40,z0,tPen\WObj:=wPaper;
    MoveL Offs(pOrigin,384.09,142.91,0.00),v40,z0,tPen\WObj:=wPaper;
    MoveL Offs(pOrigin,378.77,138.95,0.00),v40,z0,tPen\WObj:=wPaper;
    MoveL Offs(pOrigin,378.00,138.88,0.00),v40,z0,tPen\WObj:=wPaper;
    MoveL Offs(pOrigin,378.35,139.73,0.00),v40,z0,tPen\WObj:=wPaper;
    MoveL Offs(pOrigin,384.30,144.82,0.00),v40,z0,tPen\WObj:=wPaper;
    MoveL Offs(pOrigin,385.08,145.89,0.00),v40,z0,tPen\WObj:=wPaper;
    MoveL Offs(pOrigin,385.58,147.38,0.00),v40,z0,tPen\WObj:=wPaper;
    MoveL Offs(pOrigin,385.58,148.86,0.00),v40,z0,tPen\WObj:=wPaper;
    MoveL Offs(pOrigin,385.01,150.77,0.00),v40,z0,tPen\WObj:=wPaper;
    MoveL Offs(pOrigin,380.62,160.34,0.00),v40,z0,tPen\WObj:=wPaper;
    MoveL Offs(pOrigin,379.41,163.74,0.00),v40,z0,tPen\WObj:=wPaper;
    MoveL Offs(pOrigin,378.99,163.88,0.00),v40,z0,tPen\WObj:=wPaper;
    MoveL Offs(pOrigin,378.49,163.52,0.00),v40,z0,tPen\WObj:=wPaper;
    MoveL Offs(pOrigin,366.45,148.86,0.00),v40,z0,tPen\WObj:=wPaper;
    MoveL Offs(pOrigin,365.81,148.65,0.00),v40,z0,tPen\WObj:=wPaper;
    MoveL Offs(pOrigin,365.81,148.65,0.00),v40,z0,tPen\WObj:=wPaper;
    MoveL Offs(pOrigin,365.74,147.80,0.00),v40,z0,tPen\WObj:=wPaper;
    MoveL Offs(pOrigin,364.54,147.16,0.00),v40,z0,tPen\WObj:=wPaper;
    MoveL Offs(pOrigin,359.23,140.57,0.00),v40,z0,tPen\WObj:=wPaper;
    MoveL Offs(pOrigin,359.82,140.72,0.00),v40,z0,tPen\WObj:=wPaper;
    MoveL Offs(pOrigin,364.63,135.91,0.00),v40,z0,tPen\WObj:=wPaper;
    MoveL Offs(pOrigin,364.11,136.44,0.00),v40,z0,tPen\WObj:=wPaper;
    MoveL Offs(pOrigin,362.41,136.44,0.00),v40,z0,tPen\WObj:=wPaper;
    MoveL Offs(pOrigin,361.77,135.90,0.00),v40,z0,tPen\WObj:=wPaper;
    MoveL Offs(pOrigin,362.62,136.75,0.00),v40,z0,tPen\WObj:=wPaper;
    MoveL Offs(pOrigin,361.77,135.90,0.00),v40,z0,tPen\WObj:=wPaper;
    MoveL Offs(pOrigin,361.14,135.38,0.00),v40,z0,tPen\WObj:=wPaper;
    MoveL Offs(pOrigin,363.05,135.38,0.00),v40,z0,tPen\WObj:=wPaper;
    MoveL Offs(pOrigin,363.88,135.17,0.00),v40,z0,tPen\WObj:=wPaper;
    MoveL Offs(pOrigin,359.52,139.52,0.00),v40,z0,tPen\WObj:=wPaper;
    MoveL Offs(pOrigin,358.93,138.63,0.00),v40,z0,tPen\WObj:=wPaper;
    MoveL Offs(pOrigin,363.14,134.42,0.00),v40,z0,tPen\WObj:=wPaper;
    MoveL Offs(pOrigin,362.39,133.67,0.00),v40,z0,tPen\WObj:=wPaper;
    MoveL Offs(pOrigin,358.18,137.88,0.00),v40,z0,tPen\WObj:=wPaper;
    MoveL Offs(pOrigin,358.70,137.97,0.00),v40,z0,tPen\WObj:=wPaper;
    MoveL Offs(pOrigin,365.31,144.58,0.00),v40,z0,tPen\WObj:=wPaper;
    MoveL Offs(pOrigin,365.81,143.76,0.00),v40,z0,tPen\WObj:=wPaper;
    MoveL Offs(pOrigin,366.88,144.82,0.00),v40,z0,tPen\WObj:=wPaper;
    MoveL Offs(pOrigin,367.73,145.46,0.00),v40,z0,tPen\WObj:=wPaper;
    MoveL Offs(pOrigin,368.15,145.89,0.00),v40,z0,tPen\WObj:=wPaper;
    MoveL Offs(pOrigin,367.73,145.46,0.00),v40,fine,tPen\WObj:=wPaper;
    MoveL Offs(pOrigin,367.73,145.46,6.00),v60,z5,tPen\WObj:=wPaper;
    MoveL Offs(pOrigin,367.29,146.69,6.00),vTravel,z5,tPen\WObj:=wPaper;
  ENDPROC

  PROC DrawPart56()
    MoveL Offs(pOrigin,367.29,146.69,0.00),v60,z0,tPen\WObj:=wPaper;
    MoveL Offs(pOrigin,369.10,144.89,0.00),v40,z0,tPen\WObj:=wPaper;
    MoveL Offs(pOrigin,369.84,145.63,0.00),v40,z0,tPen\WObj:=wPaper;
    MoveL Offs(pOrigin,368.19,147.29,0.00),v40,z0,tPen\WObj:=wPaper;
    MoveL Offs(pOrigin,368.94,148.03,0.00),v40,z0,tPen\WObj:=wPaper;
    MoveL Offs(pOrigin,370.59,146.38,0.00),v40,z0,tPen\WObj:=wPaper;
    MoveL Offs(pOrigin,371.49,146.98,0.00),v40,z0,tPen\WObj:=wPaper;
    MoveL Offs(pOrigin,369.98,148.48,0.00),v40,z0,tPen\WObj:=wPaper;
    MoveL Offs(pOrigin,370.72,148.49,0.00),v40,z0,tPen\WObj:=wPaper;
    MoveL Offs(pOrigin,351.03,128.81,0.00),v40,z0,tPen\WObj:=wPaper;
    MoveL Offs(pOrigin,350.87,128.76,0.00),v40,z0,tPen\WObj:=wPaper;
    MoveL Offs(pOrigin,355.38,124.26,0.00),v40,z0,tPen\WObj:=wPaper;
    MoveL Offs(pOrigin,354.76,124.82,0.00),v40,z0,tPen\WObj:=wPaper;
    MoveL Offs(pOrigin,350.94,124.82,0.00),v40,z0,tPen\WObj:=wPaper;
    MoveL Offs(pOrigin,350.42,125.21,0.00),v40,z0,tPen\WObj:=wPaper;
    MoveL Offs(pOrigin,363.80,138.59,0.00),v40,z0,tPen\WObj:=wPaper;
    MoveL Offs(pOrigin,363.69,137.50,0.00),v40,z0,tPen\WObj:=wPaper;
    MoveL Offs(pOrigin,365.17,137.50,0.00),v40,z0,tPen\WObj:=wPaper;
    MoveL Offs(pOrigin,365.44,137.24,0.00),v40,z0,tPen\WObj:=wPaper;
    MoveL Offs(pOrigin,370.85,142.65,0.00),v40,z0,tPen\WObj:=wPaper;
    MoveL Offs(pOrigin,370.90,143.08,0.00),v40,z0,tPen\WObj:=wPaper;
    MoveL Offs(pOrigin,372.70,141.28,0.00),v40,z0,tPen\WObj:=wPaper;
    MoveL Offs(pOrigin,371.80,140.68,0.00),v40,z0,tPen\WObj:=wPaper;
    MoveL Offs(pOrigin,369.85,142.64,0.00),v40,z0,tPen\WObj:=wPaper;
    MoveL Offs(pOrigin,368.95,142.04,0.00),v40,z0,tPen\WObj:=wPaper;
    MoveL Offs(pOrigin,370.76,140.24,0.00),v40,z0,tPen\WObj:=wPaper;
    MoveL Offs(pOrigin,370.55,140.85,0.00),v40,z0,tPen\WObj:=wPaper;
    MoveL Offs(pOrigin,372.95,143.26,0.00),v40,z0,tPen\WObj:=wPaper;
    MoveL Offs(pOrigin,373.14,143.83,0.00),v40,z0,tPen\WObj:=wPaper;
    MoveL Offs(pOrigin,374.65,142.32,0.00),v40,z0,tPen\WObj:=wPaper;
    MoveL Offs(pOrigin,373.75,141.73,0.00),v40,z0,tPen\WObj:=wPaper;
    MoveL Offs(pOrigin,371.95,143.53,0.00),v40,fine,tPen\WObj:=wPaper;
    MoveL Offs(pOrigin,371.95,143.53,6.00),v60,z5,tPen\WObj:=wPaper;
    MoveL Offs(pOrigin,371.76,142.27,6.00),vTravel,z5,tPen\WObj:=wPaper;
    MoveL Offs(pOrigin,371.76,142.27,0.00),v60,z0,tPen\WObj:=wPaper;
    MoveL Offs(pOrigin,370.06,141.92,0.00),v40,z0,tPen\WObj:=wPaper;
    MoveL Offs(pOrigin,366.66,140.01,0.00),v40,z0,tPen\WObj:=wPaper;
    MoveL Offs(pOrigin,361.14,135.69,0.00),v40,z0,tPen\WObj:=wPaper;
    MoveL Offs(pOrigin,356.89,130.80,0.00),v40,z0,tPen\WObj:=wPaper;
    MoveL Offs(pOrigin,353.42,125.49,0.00),v40,z0,tPen\WObj:=wPaper;
    MoveL Offs(pOrigin,352.85,125.06,0.00),v40,z0,tPen\WObj:=wPaper;
    MoveL Offs(pOrigin,352.85,125.06,0.00),v40,z0,tPen\WObj:=wPaper;
    MoveL Offs(pOrigin,352.64,125.70,0.00),v40,z0,tPen\WObj:=wPaper;
    MoveL Offs(pOrigin,353.70,128.25,0.00),v40,z0,tPen\WObj:=wPaper;
    MoveL Offs(pOrigin,354.05,130.38,0.00),v40,z0,tPen\WObj:=wPaper;
    MoveL Offs(pOrigin,354.98,131.23,0.00),v40,z0,tPen\WObj:=wPaper;
    MoveL Offs(pOrigin,355.61,132.50,0.00),v40,z0,tPen\WObj:=wPaper;
    MoveL Offs(pOrigin,355.61,132.50,0.00),v40,z0,tPen\WObj:=wPaper;
    MoveL Offs(pOrigin,355.90,133.56,0.00),v40,z0,tPen\WObj:=wPaper;
    MoveL Offs(pOrigin,357.95,136.32,0.00),v40,z0,tPen\WObj:=wPaper;
    MoveL Offs(pOrigin,358.59,136.75,0.00),v40,z0,tPen\WObj:=wPaper;
    MoveL Offs(pOrigin,358.59,136.75,0.00),v40,z0,tPen\WObj:=wPaper;
    MoveL Offs(pOrigin,358.80,137.39,0.00),v40,z0,tPen\WObj:=wPaper;
    MoveL Offs(pOrigin,360.08,138.45,0.00),v40,z0,tPen\WObj:=wPaper;
    MoveL Offs(pOrigin,360.08,138.45,0.00),v40,z0,tPen\WObj:=wPaper;
    MoveL Offs(pOrigin,360.92,139.73,0.00),v40,z0,tPen\WObj:=wPaper;
    MoveL Offs(pOrigin,363.26,141.21,0.00),v40,z0,tPen\WObj:=wPaper;
    MoveL Offs(pOrigin,363.26,141.21,0.00),v40,z0,tPen\WObj:=wPaper;
    MoveL Offs(pOrigin,364.54,141.64,0.00),v40,z0,tPen\WObj:=wPaper;
    MoveL Offs(pOrigin,366.02,143.76,0.00),v40,z0,tPen\WObj:=wPaper;
    MoveL Offs(pOrigin,369.64,146.95,0.00),v40,z0,tPen\WObj:=wPaper;
    MoveL Offs(pOrigin,375.16,150.77,0.00),v40,z0,tPen\WObj:=wPaper;
    MoveL Offs(pOrigin,374.62,149.81,0.00),v40,z0,tPen\WObj:=wPaper;
    MoveL Offs(pOrigin,373.72,150.71,0.00),v40,z0,tPen\WObj:=wPaper;
    MoveL Offs(pOrigin,372.67,150.27,0.00),v40,z0,tPen\WObj:=wPaper;
    MoveL Offs(pOrigin,373.88,149.07,0.00),v40,z0,tPen\WObj:=wPaper;
    MoveL Offs(pOrigin,373.13,148.32,0.00),v40,z0,tPen\WObj:=wPaper;
    MoveL Offs(pOrigin,371.78,149.67,0.00),v40,z0,tPen\WObj:=wPaper;
    MoveL Offs(pOrigin,370.73,149.23,0.00),v40,z0,tPen\WObj:=wPaper;
    MoveL Offs(pOrigin,372.38,147.57,0.00),v40,fine,tPen\WObj:=wPaper;
    MoveL Offs(pOrigin,372.38,147.57,6.00),v60,z5,tPen\WObj:=wPaper;
    MoveL Offs(pOrigin,374.34,144.12,6.00),vTravel,z5,tPen\WObj:=wPaper;
    MoveL Offs(pOrigin,374.34,144.12,0.00),v60,z0,tPen\WObj:=wPaper;
    MoveL Offs(pOrigin,375.69,142.77,0.00),v40,z0,tPen\WObj:=wPaper;
    MoveL Offs(pOrigin,376.59,143.37,0.00),v40,z0,tPen\WObj:=wPaper;
    MoveL Offs(pOrigin,375.54,144.42,0.00),v40,fine,tPen\WObj:=wPaper;
    MoveL Offs(pOrigin,375.54,144.42,6.00),v60,z5,tPen\WObj:=wPaper;
    MoveL Offs(pOrigin,377.71,144.19,6.00),vTravel,z5,tPen\WObj:=wPaper;
    MoveL Offs(pOrigin,377.71,144.19,0.00),v60,z0,tPen\WObj:=wPaper;
    MoveL Offs(pOrigin,371.76,142.27,0.00),v40,z0,tPen\WObj:=wPaper;
    MoveL Offs(pOrigin,371.76,142.27,0.00),v40,z0,tPen\WObj:=wPaper;
    MoveL Offs(pOrigin,371.34,141.35,0.00),v40,z0,tPen\WObj:=wPaper;
    MoveL Offs(pOrigin,369.42,140.50,0.00),v40,z0,tPen\WObj:=wPaper;
    MoveL Offs(pOrigin,364.96,137.18,0.00),v40,z0,tPen\WObj:=wPaper;
    MoveL Offs(pOrigin,360.08,132.29,0.00),v40,z0,tPen\WObj:=wPaper;
    MoveL Offs(pOrigin,357.10,128.46,0.00),v40,z0,tPen\WObj:=wPaper;
    MoveL Offs(pOrigin,354.41,124.21,0.00),v40,z0,tPen\WObj:=wPaper;
    MoveL Offs(pOrigin,351.72,118.26,0.00),v40,z0,tPen\WObj:=wPaper;
    MoveL Offs(pOrigin,350.30,112.95,0.00),v40,z0,tPen\WObj:=wPaper;
    MoveL Offs(pOrigin,350.30,111.89,0.00),v40,z0,tPen\WObj:=wPaper;
    MoveL Offs(pOrigin,350.73,111.25,0.00),v40,z0,tPen\WObj:=wPaper;
    MoveL Offs(pOrigin,351.79,111.10,0.00),v40,z0,tPen\WObj:=wPaper;
    MoveL Offs(pOrigin,347.96,111.10,0.00),v40,z0,tPen\WObj:=wPaper;
    MoveL Offs(pOrigin,347.33,111.40,0.00),v40,z0,tPen\WObj:=wPaper;
    MoveL Offs(pOrigin,354.54,104.19,0.00),v40,z0,tPen\WObj:=wPaper;
    MoveL Offs(pOrigin,353.70,104.76,0.00),v40,z0,tPen\WObj:=wPaper;
    MoveL Offs(pOrigin,352.21,104.76,0.00),v40,z0,tPen\WObj:=wPaper;
    MoveL Offs(pOrigin,351.79,104.66,0.00),v40,z0,tPen\WObj:=wPaper;
    MoveL Offs(pOrigin,352.64,105.51,0.00),v40,z0,tPen\WObj:=wPaper;
    MoveL Offs(pOrigin,351.79,104.66,0.00),v40,fine,tPen\WObj:=wPaper;
    MoveL Offs(pOrigin,351.79,104.66,6.00),v60,z5,tPen\WObj:=wPaper;
    MoveL Offs(pOrigin,352.64,103.70,6.00),vTravel,z5,tPen\WObj:=wPaper;
    MoveL Offs(pOrigin,352.64,103.70,0.00),v60,z0,tPen\WObj:=wPaper;
    MoveL Offs(pOrigin,345.84,103.70,0.00),v40,z0,tPen\WObj:=wPaper;
    MoveL Offs(pOrigin,346.38,104.24,0.00),v40,z0,tPen\WObj:=wPaper;
    MoveL Offs(pOrigin,346.38,97.22,0.00),v40,z0,tPen\WObj:=wPaper;
    MoveL Offs(pOrigin,347.11,97.01,0.00),v40,z0,tPen\WObj:=wPaper;
    MoveL Offs(pOrigin,347.33,99.56,0.00),v40,fine,tPen\WObj:=wPaper;
    MoveL Offs(pOrigin,347.33,99.56,6.00),v60,z5,tPen\WObj:=wPaper;
    MoveL Offs(pOrigin,346.26,101.05,6.00),vTravel,z5,tPen\WObj:=wPaper;
    MoveL Offs(pOrigin,346.26,101.05,0.00),v60,z0,tPen\WObj:=wPaper;
    MoveL Offs(pOrigin,346.48,100.41,0.00),v40,z0,tPen\WObj:=wPaper;
    MoveL Offs(pOrigin,344.14,91.91,0.00),v40,z0,tPen\WObj:=wPaper;
    MoveL Offs(pOrigin,339.82,80.65,0.00),v40,z0,tPen\WObj:=wPaper;
    MoveL Offs(pOrigin,339.67,79.38,0.00),v40,z0,tPen\WObj:=wPaper;
    MoveL Offs(pOrigin,340.55,79.49,0.00),v40,z0,tPen\WObj:=wPaper;
    MoveL Offs(pOrigin,333.94,72.88,0.00),v40,z0,tPen\WObj:=wPaper;
    MoveL Offs(pOrigin,333.51,73.08,0.00),v40,z0,tPen\WObj:=wPaper;
    MoveL Offs(pOrigin,326.50,73.08,0.00),v40,z0,tPen\WObj:=wPaper;
    MoveL Offs(pOrigin,325.85,73.76,0.00),v40,z0,tPen\WObj:=wPaper;
  ENDPROC

  PROC DrawPart57()
    MoveL Offs(pOrigin,322.69,70.60,0.00),v40,z0,tPen\WObj:=wPaper;
    MoveL Offs(pOrigin,322.89,70.13,0.00),v40,z0,tPen\WObj:=wPaper;
    MoveL Offs(pOrigin,320.33,72.68,0.00),v40,z0,tPen\WObj:=wPaper;
    MoveL Offs(pOrigin,319.85,72.24,0.00),v40,z0,tPen\WObj:=wPaper;
    MoveL Offs(pOrigin,313.84,66.23,0.00),v40,z0,tPen\WObj:=wPaper;
    MoveL Offs(pOrigin,313.91,65.66,0.00),v40,z0,tPen\WObj:=wPaper;
    MoveL Offs(pOrigin,310.61,68.97,0.00),v40,z0,tPen\WObj:=wPaper;
    MoveL Offs(pOrigin,311.50,69.56,0.00),v40,z0,tPen\WObj:=wPaper;
    MoveL Offs(pOrigin,315.26,65.81,0.00),v40,z0,tPen\WObj:=wPaper;
    MoveL Offs(pOrigin,315.49,66.38,0.00),v40,z0,tPen\WObj:=wPaper;
    MoveL Offs(pOrigin,321.95,72.85,0.00),v40,z0,tPen\WObj:=wPaper;
    MoveL Offs(pOrigin,321.38,73.13,0.00),v40,z0,tPen\WObj:=wPaper;
    MoveL Offs(pOrigin,324.08,70.42,0.00),v40,z0,tPen\WObj:=wPaper;
    MoveL Offs(pOrigin,324.64,71.06,0.00),v40,z0,tPen\WObj:=wPaper;
    MoveL Offs(pOrigin,327.50,73.91,0.00),v40,z0,tPen\WObj:=wPaper;
    MoveL Offs(pOrigin,327.52,74.46,0.00),v40,z0,tPen\WObj:=wPaper;
    MoveL Offs(pOrigin,330.37,71.60,0.00),v40,z0,tPen\WObj:=wPaper;
    MoveL Offs(pOrigin,330.49,72.42,0.00),v40,z0,tPen\WObj:=wPaper;
    MoveL Offs(pOrigin,333.04,74.98,0.00),v40,z0,tPen\WObj:=wPaper;
    MoveL Offs(pOrigin,332.61,75.34,0.00),v40,z0,tPen\WObj:=wPaper;
    MoveL Offs(pOrigin,335.46,72.49,0.00),v40,z0,tPen\WObj:=wPaper;
    MoveL Offs(pOrigin,335.58,73.04,0.00),v40,z0,tPen\WObj:=wPaper;
    MoveL Offs(pOrigin,339.19,76.64,0.00),v40,z0,tPen\WObj:=wPaper;
    MoveL Offs(pOrigin,340.09,76.05,0.00),v40,z0,tPen\WObj:=wPaper;
    MoveL Offs(pOrigin,337.53,73.49,0.00),v40,z0,tPen\WObj:=wPaper;
    MoveL Offs(pOrigin,338.01,72.93,0.00),v40,z0,tPen\WObj:=wPaper;
    MoveL Offs(pOrigin,334.55,76.38,0.00),v40,z0,tPen\WObj:=wPaper;
    MoveL Offs(pOrigin,334.99,75.43,0.00),v40,z0,tPen\WObj:=wPaper;
    MoveL Offs(pOrigin,332.14,72.58,0.00),v40,z0,tPen\WObj:=wPaper;
    MoveL Offs(pOrigin,331.57,71.90,0.00),v40,z0,tPen\WObj:=wPaper;
    MoveL Offs(pOrigin,328.71,74.75,0.00),v40,z0,tPen\WObj:=wPaper;
    MoveL Offs(pOrigin,329.45,74.37,0.00),v40,z0,tPen\WObj:=wPaper;
    MoveL Offs(pOrigin,326.59,71.51,0.00),v40,z0,tPen\WObj:=wPaper;
    MoveL Offs(pOrigin,326.48,71.02,0.00),v40,z0,tPen\WObj:=wPaper;
    MoveL Offs(pOrigin,323.77,73.72,0.00),v40,z0,tPen\WObj:=wPaper;
    MoveL Offs(pOrigin,323.90,73.30,0.00),v40,z0,tPen\WObj:=wPaper;
    MoveL Offs(pOrigin,320.60,70.00,0.00),v40,z0,tPen\WObj:=wPaper;
    MoveL Offs(pOrigin,319.84,69.24,0.00),v40,z0,tPen\WObj:=wPaper;
    MoveL Offs(pOrigin,317.44,66.84,0.00),v40,z0,tPen\WObj:=wPaper;
    MoveL Offs(pOrigin,317.96,66.10,0.00),v40,z0,tPen\WObj:=wPaper;
    MoveL Offs(pOrigin,313.60,70.46,0.00),v40,z0,tPen\WObj:=wPaper;
    MoveL Offs(pOrigin,313.33,69.60,0.00),v40,z0,tPen\WObj:=wPaper;
    MoveL Offs(pOrigin,313.75,69.81,0.00),v40,z0,tPen\WObj:=wPaper;
    MoveL Offs(pOrigin,313.33,69.60,0.00),v40,z0,tPen\WObj:=wPaper;
    MoveL Offs(pOrigin,312.80,69.67,0.00),v40,z0,tPen\WObj:=wPaper;
    MoveL Offs(pOrigin,302.74,59.60,0.00),v40,z0,tPen\WObj:=wPaper;
    MoveL Offs(pOrigin,302.70,58.96,0.00),v40,z0,tPen\WObj:=wPaper;
    MoveL Offs(pOrigin,297.74,63.91,0.00),v40,z0,tPen\WObj:=wPaper;
    MoveL Offs(pOrigin,297.81,63.63,0.00),v40,z0,tPen\WObj:=wPaper;
    MoveL Offs(pOrigin,295.85,61.68,0.00),v40,fine,tPen\WObj:=wPaper;
    MoveL Offs(pOrigin,295.85,61.68,6.00),v60,z5,tPen\WObj:=wPaper;
    MoveL Offs(pOrigin,294.66,61.98,6.00),vTravel,z5,tPen\WObj:=wPaper;
    MoveL Offs(pOrigin,294.66,61.98,0.00),v60,z0,tPen\WObj:=wPaper;
    MoveL Offs(pOrigin,296.31,63.63,0.00),v40,z0,tPen\WObj:=wPaper;
    MoveL Offs(pOrigin,295.26,64.08,0.00),v40,z0,tPen\WObj:=wPaper;
    MoveL Offs(pOrigin,293.46,62.27,0.00),v40,z0,tPen\WObj:=wPaper;
    MoveL Offs(pOrigin,294.20,62.52,0.00),v40,z0,tPen\WObj:=wPaper;
    MoveL Offs(pOrigin,305.04,62.52,0.00),v40,fine,tPen\WObj:=wPaper;
    MoveL Offs(pOrigin,305.04,62.52,6.00),v60,z5,tPen\WObj:=wPaper;
    MoveL Offs(pOrigin,305.68,64.63,6.00),vTravel,z5,tPen\WObj:=wPaper;
    MoveL Offs(pOrigin,305.68,64.63,0.00),v60,z0,tPen\WObj:=wPaper;
    MoveL Offs(pOrigin,301.42,64.63,0.00),v40,fine,tPen\WObj:=wPaper;
    MoveL Offs(pOrigin,301.42,64.63,6.00),v60,z5,tPen\WObj:=wPaper;
    MoveL Offs(pOrigin,301.63,66.00,6.00),vTravel,z5,tPen\WObj:=wPaper;
    MoveL Offs(pOrigin,301.63,66.00,0.00),v60,z0,tPen\WObj:=wPaper;
    MoveL Offs(pOrigin,308.99,58.64,0.00),v40,z0,tPen\WObj:=wPaper;
    MoveL Offs(pOrigin,308.43,59.32,0.00),v40,z0,tPen\WObj:=wPaper;
    MoveL Offs(pOrigin,312.79,63.68,0.00),v40,z0,tPen\WObj:=wPaper;
    MoveL Offs(pOrigin,312.59,62.59,0.00),v40,z0,tPen\WObj:=wPaper;
    MoveL Offs(pOrigin,312.59,61.52,0.00),v40,z0,tPen\WObj:=wPaper;
    MoveL Offs(pOrigin,313.11,61.74,0.00),v40,z0,tPen\WObj:=wPaper;
    MoveL Offs(pOrigin,311.41,61.53,0.00),v40,z0,tPen\WObj:=wPaper;
    MoveL Offs(pOrigin,311.53,61.10,0.00),v40,z0,tPen\WObj:=wPaper;
    MoveL Offs(pOrigin,311.53,63.01,0.00),v40,z0,tPen\WObj:=wPaper;
    MoveL Offs(pOrigin,310.48,63.22,0.00),v40,z0,tPen\WObj:=wPaper;
    MoveL Offs(pOrigin,310.48,60.68,0.00),v40,z0,tPen\WObj:=wPaper;
    MoveL Offs(pOrigin,310.38,59.78,0.00),v40,z0,tPen\WObj:=wPaper;
    MoveL Offs(pOrigin,313.83,63.23,0.00),v40,z0,tPen\WObj:=wPaper;
    MoveL Offs(pOrigin,314.52,63.56,0.00),v40,z0,tPen\WObj:=wPaper;
    MoveL Offs(pOrigin,322.33,55.75,0.00),v40,z0,tPen\WObj:=wPaper;
    MoveL Offs(pOrigin,322.05,55.02,0.00),v40,z0,tPen\WObj:=wPaper;
    MoveL Offs(pOrigin,319.94,52.92,0.00),v40,z0,tPen\WObj:=wPaper;
    MoveL Offs(pOrigin,320.54,52.02,0.00),v40,z0,tPen\WObj:=wPaper;
    MoveL Offs(pOrigin,322.64,54.12,0.00),v40,z0,tPen\WObj:=wPaper;
    MoveL Offs(pOrigin,322.04,54.07,0.00),v40,z0,tPen\WObj:=wPaper;
    MoveL Offs(pOrigin,320.55,54.07,0.00),v40,z0,tPen\WObj:=wPaper;
    MoveL Offs(pOrigin,319.65,54.11,0.00),v40,z0,tPen\WObj:=wPaper;
    MoveL Offs(pOrigin,321.60,56.07,0.00),v40,z0,tPen\WObj:=wPaper;
    MoveL Offs(pOrigin,321.19,56.21,0.00),v40,z0,tPen\WObj:=wPaper;
    MoveL Offs(pOrigin,320.98,56.64,0.00),v40,z0,tPen\WObj:=wPaper;
    MoveL Offs(pOrigin,321.19,56.21,0.00),v40,z0,tPen\WObj:=wPaper;
    MoveL Offs(pOrigin,320.98,56.18,0.00),v40,z0,tPen\WObj:=wPaper;
    MoveL Offs(pOrigin,319.49,56.18,0.00),v40,fine,tPen\WObj:=wPaper;
    MoveL Offs(pOrigin,319.49,56.18,6.00),v60,z5,tPen\WObj:=wPaper;
    MoveL Offs(pOrigin,318.85,57.24,6.00),vTravel,z5,tPen\WObj:=wPaper;
    MoveL Offs(pOrigin,318.85,57.24,0.00),v60,z0,tPen\WObj:=wPaper;
    MoveL Offs(pOrigin,320.34,57.24,0.00),v40,z0,tPen\WObj:=wPaper;
    MoveL Offs(pOrigin,320.56,58.01,0.00),v40,z0,tPen\WObj:=wPaper;
    MoveL Offs(pOrigin,318.30,55.76,0.00),v40,z0,tPen\WObj:=wPaper;
    MoveL Offs(pOrigin,319.05,55.01,0.00),v40,z0,tPen\WObj:=wPaper;
    MoveL Offs(pOrigin,321.15,57.11,0.00),v40,fine,tPen\WObj:=wPaper;
    MoveL Offs(pOrigin,321.15,57.11,6.00),v60,z5,tPen\WObj:=wPaper;
    MoveL Offs(pOrigin,321.40,55.13,6.00),vTravel,z5,tPen\WObj:=wPaper;
    MoveL Offs(pOrigin,321.40,55.13,0.00),v60,z0,tPen\WObj:=wPaper;
    MoveL Offs(pOrigin,320.12,55.13,0.00),v40,fine,tPen\WObj:=wPaper;
    MoveL Offs(pOrigin,320.12,55.13,6.00),v60,z5,tPen\WObj:=wPaper;
    MoveL Offs(pOrigin,321.83,54.94,6.00),vTravel,z5,tPen\WObj:=wPaper;
    MoveL Offs(pOrigin,321.83,54.94,0.00),v60,z0,tPen\WObj:=wPaper;
    MoveL Offs(pOrigin,321.61,55.36,0.00),v40,z0,tPen\WObj:=wPaper;
    MoveL Offs(pOrigin,321.83,54.94,0.00),v40,fine,tPen\WObj:=wPaper;
    MoveL Offs(pOrigin,321.83,54.94,6.00),v60,z5,tPen\WObj:=wPaper;
    MoveL Offs(pOrigin,323.54,53.05,6.00),vTravel,z5,tPen\WObj:=wPaper;
    MoveL Offs(pOrigin,323.54,53.05,0.00),v60,z0,tPen\WObj:=wPaper;
    MoveL Offs(pOrigin,308.81,67.78,0.00),v40,z0,tPen\WObj:=wPaper;
    MoveL Offs(pOrigin,308.44,66.74,0.00),v40,z0,tPen\WObj:=wPaper;
    MoveL Offs(pOrigin,314.60,66.74,0.00),v40,z0,tPen\WObj:=wPaper;
    MoveL Offs(pOrigin,314.70,67.47,0.00),v40,z0,tPen\WObj:=wPaper;
    MoveL Offs(pOrigin,314.70,69.18,0.00),v40,z0,tPen\WObj:=wPaper;
    MoveL Offs(pOrigin,315.02,69.91,0.00),v40,z0,tPen\WObj:=wPaper;
    MoveL Offs(pOrigin,318.42,69.91,0.00),v40,z0,tPen\WObj:=wPaper;
  ENDPROC

  PROC DrawPart58()
    MoveL Offs(pOrigin,318.00,70.97,0.00),v40,z0,tPen\WObj:=wPaper;
    MoveL Offs(pOrigin,322.04,70.97,0.00),v40,z0,tPen\WObj:=wPaper;
    MoveL Offs(pOrigin,321.61,72.02,0.00),v40,z0,tPen\WObj:=wPaper;
    MoveL Offs(pOrigin,326.92,72.02,0.00),v40,z0,tPen\WObj:=wPaper;
    MoveL Offs(pOrigin,327.68,71.31,0.00),v40,z0,tPen\WObj:=wPaper;
    MoveL Offs(pOrigin,325.12,73.87,0.00),v40,z0,tPen\WObj:=wPaper;
    MoveL Offs(pOrigin,326.17,74.31,0.00),v40,z0,tPen\WObj:=wPaper;
    MoveL Offs(pOrigin,329.02,71.46,0.00),v40,z0,tPen\WObj:=wPaper;
    MoveL Offs(pOrigin,328.54,71.97,0.00),v40,z0,tPen\WObj:=wPaper;
    MoveL Offs(pOrigin,331.09,74.52,0.00),v40,z0,tPen\WObj:=wPaper;
    MoveL Offs(pOrigin,331.26,75.20,0.00),v40,z0,tPen\WObj:=wPaper;
    MoveL Offs(pOrigin,334.11,72.34,0.00),v40,fine,tPen\WObj:=wPaper;
    MoveL Offs(pOrigin,334.11,72.34,6.00),v60,z5,tPen\WObj:=wPaper;
    MoveL Offs(pOrigin,332.92,72.05,6.00),vTravel,z5,tPen\WObj:=wPaper;
    MoveL Offs(pOrigin,332.92,72.05,0.00),v60,z0,tPen\WObj:=wPaper;
    MoveL Offs(pOrigin,330.06,74.90,0.00),v40,fine,tPen\WObj:=wPaper;
    MoveL Offs(pOrigin,330.06,74.90,6.00),v60,z5,tPen\WObj:=wPaper;
    MoveL Offs(pOrigin,332.45,74.14,6.00),vTravel,z5,tPen\WObj:=wPaper;
    MoveL Offs(pOrigin,332.45,74.14,0.00),v60,z0,tPen\WObj:=wPaper;
    MoveL Offs(pOrigin,341.38,74.14,0.00),v40,z0,tPen\WObj:=wPaper;
    MoveL Offs(pOrigin,340.68,73.65,0.00),v40,z0,tPen\WObj:=wPaper;
    MoveL Offs(pOrigin,343.53,76.51,0.00),v40,z0,tPen\WObj:=wPaper;
    MoveL Offs(pOrigin,343.09,76.81,0.00),v40,z0,tPen\WObj:=wPaper;
    MoveL Offs(pOrigin,349.40,70.50,0.00),v40,z0,tPen\WObj:=wPaper;
    MoveL Offs(pOrigin,350.11,71.13,0.00),v40,z0,tPen\WObj:=wPaper;
    MoveL Offs(pOrigin,350.86,71.89,0.00),v40,z0,tPen\WObj:=wPaper;
    MoveL Offs(pOrigin,350.29,72.59,0.00),v40,z0,tPen\WObj:=wPaper;
    MoveL Offs(pOrigin,353.60,69.29,0.00),v40,z0,tPen\WObj:=wPaper;
    MoveL Offs(pOrigin,353.55,70.10,0.00),v40,z0,tPen\WObj:=wPaper;
    MoveL Offs(pOrigin,354.45,71.00,0.00),v40,z0,tPen\WObj:=wPaper;
    MoveL Offs(pOrigin,354.49,71.38,0.00),v40,z0,tPen\WObj:=wPaper;
    MoveL Offs(pOrigin,357.95,67.92,0.00),v40,z0,tPen\WObj:=wPaper;
    MoveL Offs(pOrigin,358.19,68.76,0.00),v40,z0,tPen\WObj:=wPaper;
    MoveL Offs(pOrigin,358.94,69.51,0.00),v40,z0,tPen\WObj:=wPaper;
    MoveL Offs(pOrigin,358.69,70.17,0.00),v40,z0,tPen\WObj:=wPaper;
    MoveL Offs(pOrigin,363.05,65.81,0.00),v40,z0,tPen\WObj:=wPaper;
    MoveL Offs(pOrigin,363.28,66.38,0.00),v40,z0,tPen\WObj:=wPaper;
    MoveL Offs(pOrigin,364.18,67.28,0.00),v40,z0,tPen\WObj:=wPaper;
    MoveL Offs(pOrigin,363.64,68.21,0.00),v40,z0,tPen\WObj:=wPaper;
    MoveL Offs(pOrigin,369.65,62.20,0.00),v40,z0,tPen\WObj:=wPaper;
    MoveL Offs(pOrigin,370.16,62.81,0.00),v40,z0,tPen\WObj:=wPaper;
    MoveL Offs(pOrigin,370.91,63.56,0.00),v40,fine,tPen\WObj:=wPaper;
    MoveL Offs(pOrigin,370.91,63.56,6.00),v60,z5,tPen\WObj:=wPaper;
    MoveL Offs(pOrigin,366.05,64.30,6.00),vTravel,z5,tPen\WObj:=wPaper;
    MoveL Offs(pOrigin,366.05,64.30,0.00),v60,z0,tPen\WObj:=wPaper;
    MoveL Offs(pOrigin,361.09,69.26,0.00),v40,z0,tPen\WObj:=wPaper;
    MoveL Offs(pOrigin,361.19,68.77,0.00),v40,z0,tPen\WObj:=wPaper;
    MoveL Offs(pOrigin,360.29,67.87,0.00),v40,z0,tPen\WObj:=wPaper;
    MoveL Offs(pOrigin,360.50,66.87,0.00),v40,z0,tPen\WObj:=wPaper;
    MoveL Offs(pOrigin,356.29,71.08,0.00),v40,z0,tPen\WObj:=wPaper;
    MoveL Offs(pOrigin,355.65,70.70,0.00),v40,z0,tPen\WObj:=wPaper;
    MoveL Offs(pOrigin,354.90,69.95,0.00),v40,z0,tPen\WObj:=wPaper;
    MoveL Offs(pOrigin,355.95,69.50,0.00),v40,z0,tPen\WObj:=wPaper;
    MoveL Offs(pOrigin,356.85,70.41,0.00),v40,z0,tPen\WObj:=wPaper;
    MoveL Offs(pOrigin,357.89,69.96,0.00),v40,z0,tPen\WObj:=wPaper;
    MoveL Offs(pOrigin,356.99,69.06,0.00),v40,fine,tPen\WObj:=wPaper;
    MoveL Offs(pOrigin,356.99,69.06,6.00),v60,z5,tPen\WObj:=wPaper;
    MoveL Offs(pOrigin,355.70,68.68,6.00),vTravel,z5,tPen\WObj:=wPaper;
    MoveL Offs(pOrigin,355.70,68.68,0.00),v60,z0,tPen\WObj:=wPaper;
    MoveL Offs(pOrigin,352.24,72.14,0.00),v40,fine,tPen\WObj:=wPaper;
    MoveL Offs(pOrigin,352.24,72.14,6.00),v60,z5,tPen\WObj:=wPaper;
    MoveL Offs(pOrigin,353.41,71.44,6.00),vTravel,z5,tPen\WObj:=wPaper;
    MoveL Offs(pOrigin,353.41,71.44,0.00),v60,z0,tPen\WObj:=wPaper;
    MoveL Offs(pOrigin,352.50,70.54,0.00),v40,z0,tPen\WObj:=wPaper;
    MoveL Offs(pOrigin,351.50,69.89,0.00),v40,z0,tPen\WObj:=wPaper;
    MoveL Offs(pOrigin,348.49,72.90,0.00),v40,fine,tPen\WObj:=wPaper;
    MoveL Offs(pOrigin,348.49,72.90,6.00),v60,z5,tPen\WObj:=wPaper;
    MoveL Offs(pOrigin,348.79,74.09,6.00),vTravel,z5,tPen\WObj:=wPaper;
    MoveL Offs(pOrigin,348.79,74.09,0.00),v60,z0,tPen\WObj:=wPaper;
    MoveL Offs(pOrigin,345.63,77.25,0.00),v40,z0,tPen\WObj:=wPaper;
    MoveL Offs(pOrigin,345.48,76.96,0.00),v40,z0,tPen\WObj:=wPaper;
    MoveL Offs(pOrigin,342.48,73.96,0.00),v40,fine,tPen\WObj:=wPaper;
    MoveL Offs(pOrigin,342.48,73.96,6.00),v60,z5,tPen\WObj:=wPaper;
    MoveL Offs(pOrigin,344.13,74.11,6.00),vTravel,z5,tPen\WObj:=wPaper;
    MoveL Offs(pOrigin,344.13,74.11,0.00),v60,z0,tPen\WObj:=wPaper;
    MoveL Offs(pOrigin,349.39,79.37,0.00),v40,z0,tPen\WObj:=wPaper;
    MoveL Offs(pOrigin,349.02,79.42,0.00),v40,z0,tPen\WObj:=wPaper;
    MoveL Offs(pOrigin,347.54,79.42,0.00),v40,z0,tPen\WObj:=wPaper;
    MoveL Offs(pOrigin,346.99,79.96,0.00),v40,z0,tPen\WObj:=wPaper;
    MoveL Offs(pOrigin,349.85,82.82,0.00),v40,z0,tPen\WObj:=wPaper;
    MoveL Offs(pOrigin,349.45,82.58,0.00),v40,z0,tPen\WObj:=wPaper;
    MoveL Offs(pOrigin,347.96,82.58,0.00),v40,z0,tPen\WObj:=wPaper;
    MoveL Offs(pOrigin,348.49,82.14,0.00),v40,z0,tPen\WObj:=wPaper;
    MoveL Offs(pOrigin,348.49,81.08,0.00),v40,z0,tPen\WObj:=wPaper;
    MoveL Offs(pOrigin,349.02,80.47,0.00),v40,z0,tPen\WObj:=wPaper;
    MoveL Offs(pOrigin,347.75,80.47,0.00),v40,z0,tPen\WObj:=wPaper;
    MoveL Offs(pOrigin,347.75,81.53,0.00),v40,z0,tPen\WObj:=wPaper;
    MoveL Offs(pOrigin,349.24,81.53,0.00),v40,z0,tPen\WObj:=wPaper;
    MoveL Offs(pOrigin,349.54,81.02,0.00),v40,z0,tPen\WObj:=wPaper;
    MoveL Offs(pOrigin,346.53,78.01,0.00),v40,z0,tPen\WObj:=wPaper;
    MoveL Offs(pOrigin,346.08,78.30,0.00),v40,z0,tPen\WObj:=wPaper;
    MoveL Offs(pOrigin,349.99,74.39,0.00),v40,z0,tPen\WObj:=wPaper;
    MoveL Offs(pOrigin,349.52,75.03,0.00),v40,z0,tPen\WObj:=wPaper;
    MoveL Offs(pOrigin,354.33,79.84,0.00),v40,z0,tPen\WObj:=wPaper;
    MoveL Offs(pOrigin,353.91,79.42,0.00),v40,z0,tPen\WObj:=wPaper;
    MoveL Offs(pOrigin,352.21,79.42,0.00),v40,z0,tPen\WObj:=wPaper;
    MoveL Offs(pOrigin,351.63,80.13,0.00),v40,z0,tPen\WObj:=wPaper;
    MoveL Offs(pOrigin,353.89,82.38,0.00),v40,z0,tPen\WObj:=wPaper;
    MoveL Offs(pOrigin,353.49,82.58,0.00),v40,z0,tPen\WObj:=wPaper;
    MoveL Offs(pOrigin,351.79,82.58,0.00),v40,z0,tPen\WObj:=wPaper;
    MoveL Offs(pOrigin,351.19,82.67,0.00),v40,z0,tPen\WObj:=wPaper;
    MoveL Offs(pOrigin,353.60,85.08,0.00),v40,z0,tPen\WObj:=wPaper;
    MoveL Offs(pOrigin,354.00,85.31,0.00),v40,z0,tPen\WObj:=wPaper;
    MoveL Offs(pOrigin,347.54,91.77,0.00),v40,z0,tPen\WObj:=wPaper;
    MoveL Offs(pOrigin,348.60,92.09,0.00),v40,z0,tPen\WObj:=wPaper;
    MoveL Offs(pOrigin,353.06,92.09,0.00),v40,z0,tPen\WObj:=wPaper;
    MoveL Offs(pOrigin,352.42,91.91,0.00),v40,z0,tPen\WObj:=wPaper;
    MoveL Offs(pOrigin,352.42,91.28,0.00),v40,z0,tPen\WObj:=wPaper;
    MoveL Offs(pOrigin,353.27,91.28,0.00),v40,z0,tPen\WObj:=wPaper;
    MoveL Offs(pOrigin,354.13,91.15,0.00),v40,z0,tPen\WObj:=wPaper;
    MoveL Offs(pOrigin,344.06,101.22,0.00),v40,z0,tPen\WObj:=wPaper;
    MoveL Offs(pOrigin,344.51,101.38,0.00),v40,z0,tPen\WObj:=wPaper;
    MoveL Offs(pOrigin,357.88,114.75,0.00),v40,z0,tPen\WObj:=wPaper;
    MoveL Offs(pOrigin,357.35,114.81,0.00),v40,z0,tPen\WObj:=wPaper;
    MoveL Offs(pOrigin,359.31,112.86,0.00),v40,z0,tPen\WObj:=wPaper;
    MoveL Offs(pOrigin,359.83,113.71,0.00),v40,z0,tPen\WObj:=wPaper;
    MoveL Offs(pOrigin,362.98,116.86,0.00),v40,z0,tPen\WObj:=wPaper;
    MoveL Offs(pOrigin,362.29,117.34,0.00),v40,z0,tPen\WObj:=wPaper;
    MoveL Offs(pOrigin,364.09,115.54,0.00),v40,z0,tPen\WObj:=wPaper;
    MoveL Offs(pOrigin,363.73,116.12,0.00),v40,z0,tPen\WObj:=wPaper;
  ENDPROC

  PROC DrawPart59()
    MoveL Offs(pOrigin,364.93,117.32,0.00),v40,z0,tPen\WObj:=wPaper;
    MoveL Offs(pOrigin,364.68,117.94,0.00),v40,z0,tPen\WObj:=wPaper;
    MoveL Offs(pOrigin,366.19,116.43,0.00),v40,z0,tPen\WObj:=wPaper;
    MoveL Offs(pOrigin,365.14,115.99,0.00),v40,z0,tPen\WObj:=wPaper;
    MoveL Offs(pOrigin,363.49,117.64,0.00),v40,fine,tPen\WObj:=wPaper;
    MoveL Offs(pOrigin,363.49,117.64,6.00),v60,z5,tPen\WObj:=wPaper;
    MoveL Offs(pOrigin,361.39,116.75,6.00),vTravel,z5,tPen\WObj:=wPaper;
    MoveL Offs(pOrigin,361.39,116.75,0.00),v60,z0,tPen\WObj:=wPaper;
    MoveL Offs(pOrigin,363.20,114.95,0.00),v40,z0,tPen\WObj:=wPaper;
    MoveL Offs(pOrigin,362.15,114.50,0.00),v40,z0,tPen\WObj:=wPaper;
    MoveL Offs(pOrigin,360.34,116.30,0.00),v40,z0,tPen\WObj:=wPaper;
    MoveL Offs(pOrigin,360.58,115.96,0.00),v40,z0,tPen\WObj:=wPaper;
    MoveL Offs(pOrigin,353.67,109.04,0.00),v40,z0,tPen\WObj:=wPaper;
    MoveL Offs(pOrigin,353.49,109.55,0.00),v40,z0,tPen\WObj:=wPaper;
    MoveL Offs(pOrigin,354.34,110.40,0.00),v40,z0,tPen\WObj:=wPaper;
    MoveL Offs(pOrigin,353.49,109.55,0.00),v40,z0,tPen\WObj:=wPaper;
    MoveL Offs(pOrigin,354.12,110.04,0.00),v40,z0,tPen\WObj:=wPaper;
    MoveL Offs(pOrigin,347.54,110.04,0.00),v40,z0,tPen\WObj:=wPaper;
    MoveL Offs(pOrigin,346.93,109.77,0.00),v40,z0,tPen\WObj:=wPaper;
    MoveL Offs(pOrigin,362.56,125.40,0.00),v40,z0,tPen\WObj:=wPaper;
    MoveL Offs(pOrigin,362.41,124.85,0.00),v40,z0,tPen\WObj:=wPaper;
    MoveL Offs(pOrigin,363.26,125.49,0.00),v40,z0,tPen\WObj:=wPaper;
    MoveL Offs(pOrigin,362.41,124.85,0.00),v40,z0,tPen\WObj:=wPaper;
    MoveL Offs(pOrigin,361.66,125.44,0.00),v40,z0,tPen\WObj:=wPaper;
    MoveL Offs(pOrigin,363.17,123.93,0.00),v40,z0,tPen\WObj:=wPaper;
    MoveL Offs(pOrigin,362.42,123.19,0.00),v40,z0,tPen\WObj:=wPaper;
    MoveL Offs(pOrigin,360.92,124.69,0.00),v40,z0,tPen\WObj:=wPaper;
    MoveL Offs(pOrigin,360.02,124.09,0.00),v40,z0,tPen\WObj:=wPaper;
    MoveL Offs(pOrigin,361.52,122.59,0.00),v40,z0,tPen\WObj:=wPaper;
    MoveL Offs(pOrigin,360.78,121.84,0.00),v40,z0,tPen\WObj:=wPaper;
    MoveL Offs(pOrigin,359.12,123.50,0.00),v40,z0,tPen\WObj:=wPaper;
    MoveL Offs(pOrigin,358.38,122.75,0.00),v40,z0,tPen\WObj:=wPaper;
    MoveL Offs(pOrigin,360.03,121.10,0.00),v40,z0,tPen\WObj:=wPaper;
    MoveL Offs(pOrigin,359.43,120.20,0.00),v40,z0,tPen\WObj:=wPaper;
    MoveL Offs(pOrigin,357.63,122.00,0.00),v40,z0,tPen\WObj:=wPaper;
    MoveL Offs(pOrigin,357.03,121.11,0.00),v40,z0,tPen\WObj:=wPaper;
    MoveL Offs(pOrigin,358.69,119.45,0.00),v40,z0,tPen\WObj:=wPaper;
    MoveL Offs(pOrigin,357.94,118.71,0.00),v40,z0,tPen\WObj:=wPaper;
    MoveL Offs(pOrigin,356.14,120.51,0.00),v40,z0,tPen\WObj:=wPaper;
    MoveL Offs(pOrigin,355.39,119.76,0.00),v40,z0,tPen\WObj:=wPaper;
    MoveL Offs(pOrigin,357.19,117.96,0.00),v40,z0,tPen\WObj:=wPaper;
    MoveL Offs(pOrigin,356.84,118.19,0.00),v40,z0,tPen\WObj:=wPaper;
    MoveL Offs(pOrigin,346.03,107.37,0.00),v40,z0,tPen\WObj:=wPaper;
    MoveL Offs(pOrigin,345.84,106.91,0.00),v40,z0,tPen\WObj:=wPaper;
    MoveL Offs(pOrigin,351.55,101.20,0.00),v40,z0,tPen\WObj:=wPaper;
    MoveL Offs(pOrigin,350.72,101.59,0.00),v40,z0,tPen\WObj:=wPaper;
    MoveL Offs(pOrigin,345.20,101.59,0.00),v40,z0,tPen\WObj:=wPaper;
    MoveL Offs(pOrigin,345.41,102.65,0.00),v40,z0,tPen\WObj:=wPaper;
    MoveL Offs(pOrigin,351.58,102.65,0.00),v40,z0,tPen\WObj:=wPaper;
    MoveL Offs(pOrigin,352.00,103.18,0.00),v40,z0,tPen\WObj:=wPaper;
    MoveL Offs(pOrigin,352.85,104.03,0.00),v40,z0,tPen\WObj:=wPaper;
    MoveL Offs(pOrigin,352.00,103.18,0.00),v40,z0,tPen\WObj:=wPaper;
    MoveL Offs(pOrigin,352.90,102.84,0.00),v40,z0,tPen\WObj:=wPaper;
    MoveL Offs(pOrigin,346.43,109.30,0.00),v40,z0,tPen\WObj:=wPaper;
    MoveL Offs(pOrigin,347.33,108.98,0.00),v40,z0,tPen\WObj:=wPaper;
    MoveL Offs(pOrigin,352.85,108.98,0.00),v40,fine,tPen\WObj:=wPaper;
    MoveL Offs(pOrigin,352.85,108.98,6.00),v60,z5,tPen\WObj:=wPaper;
    MoveL Offs(pOrigin,352.00,107.93,6.00),vTravel,z5,tPen\WObj:=wPaper;
    MoveL Offs(pOrigin,352.00,107.93,0.00),v60,z0,tPen\WObj:=wPaper;
    MoveL Offs(pOrigin,346.90,107.93,0.00),v40,z0,tPen\WObj:=wPaper;
    MoveL Offs(pOrigin,347.44,108.49,0.00),v40,z0,tPen\WObj:=wPaper;
    MoveL Offs(pOrigin,347.44,97.01,0.00),v40,z0,tPen\WObj:=wPaper;
    MoveL Offs(pOrigin,347.11,97.01,0.00),v40,z0,tPen\WObj:=wPaper;
    MoveL Offs(pOrigin,348.46,94.68,0.00),v40,z0,tPen\WObj:=wPaper;
    MoveL Offs(pOrigin,348.81,92.76,0.00),v40,z0,tPen\WObj:=wPaper;
    MoveL Offs(pOrigin,348.17,84.26,0.00),v40,z0,tPen\WObj:=wPaper;
    MoveL Offs(pOrigin,346.90,76.82,0.00),v40,z0,tPen\WObj:=wPaper;
    MoveL Offs(pOrigin,346.26,76.40,0.00),v40,z0,tPen\WObj:=wPaper;
    MoveL Offs(pOrigin,339.04,75.34,0.00),v40,z0,tPen\WObj:=wPaper;
    MoveL Offs(pOrigin,337.98,75.76,0.00),v40,z0,tPen\WObj:=wPaper;
    MoveL Offs(pOrigin,337.98,75.76,0.00),v40,z0,tPen\WObj:=wPaper;
    MoveL Offs(pOrigin,339.39,78.74,0.00),v40,z0,tPen\WObj:=wPaper;
    MoveL Offs(pOrigin,340.45,79.80,0.00),v40,z0,tPen\WObj:=wPaper;
    MoveL Offs(pOrigin,342.30,83.84,0.00),v40,z0,tPen\WObj:=wPaper;
    MoveL Offs(pOrigin,347.11,97.01,0.00),v40,fine,tPen\WObj:=wPaper;
    MoveL Offs(pOrigin,347.11,97.01,6.00),v60,z5,tPen\WObj:=wPaper;
    MoveL Offs(pOrigin,346.48,95.26,6.00),vTravel,z5,tPen\WObj:=wPaper;
    MoveL Offs(pOrigin,346.48,95.26,0.00),v60,z0,tPen\WObj:=wPaper;
    MoveL Offs(pOrigin,344.99,95.26,0.00),v40,z0,tPen\WObj:=wPaper;
    MoveL Offs(pOrigin,344.78,94.20,0.00),v40,z0,tPen\WObj:=wPaper;
    MoveL Offs(pOrigin,346.05,94.20,0.00),v40,z0,tPen\WObj:=wPaper;
    MoveL Offs(pOrigin,345.62,93.14,0.00),v40,z0,tPen\WObj:=wPaper;
    MoveL Offs(pOrigin,344.56,93.14,0.00),v40,z0,tPen\WObj:=wPaper;
    MoveL Offs(pOrigin,343.43,92.83,0.00),v40,z0,tPen\WObj:=wPaper;
    MoveL Offs(pOrigin,349.60,99.00,0.00),v40,z0,tPen\WObj:=wPaper;
    MoveL Offs(pOrigin,349.45,99.48,0.00),v40,z0,tPen\WObj:=wPaper;
    MoveL Offs(pOrigin,344.56,99.48,0.00),v40,z0,tPen\WObj:=wPaper;
    MoveL Offs(pOrigin,344.78,100.54,0.00),v40,z0,tPen\WObj:=wPaper;
    MoveL Offs(pOrigin,350.09,100.54,0.00),v40,z0,tPen\WObj:=wPaper;
    MoveL Offs(pOrigin,349.66,100.41,0.00),v40,z0,tPen\WObj:=wPaper;
    MoveL Offs(pOrigin,350.30,101.26,0.00),v40,z0,tPen\WObj:=wPaper;
    MoveL Offs(pOrigin,349.66,100.41,0.00),v40,z0,tPen\WObj:=wPaper;
    MoveL Offs(pOrigin,349.55,100.84,0.00),v40,z0,tPen\WObj:=wPaper;
    MoveL Offs(pOrigin,349.55,103.18,0.00),v40,z0,tPen\WObj:=wPaper;
    MoveL Offs(pOrigin,350.30,103.18,0.00),v40,z0,tPen\WObj:=wPaper;
    MoveL Offs(pOrigin,351.15,104.03,0.00),v40,z0,tPen\WObj:=wPaper;
    MoveL Offs(pOrigin,350.30,103.18,0.00),v40,fine,tPen\WObj:=wPaper;
    MoveL Offs(pOrigin,350.30,103.18,6.00),v60,z5,tPen\WObj:=wPaper;
    MoveL Offs(pOrigin,350.51,101.69,6.00),vTravel,z5,tPen\WObj:=wPaper;
    MoveL Offs(pOrigin,350.51,101.69,0.00),v60,z0,tPen\WObj:=wPaper;
    MoveL Offs(pOrigin,351.36,102.54,0.00),v40,z0,tPen\WObj:=wPaper;
    MoveL Offs(pOrigin,350.51,101.69,0.00),v40,fine,tPen\WObj:=wPaper;
    MoveL Offs(pOrigin,350.51,101.69,6.00),v60,z5,tPen\WObj:=wPaper;
    MoveL Offs(pOrigin,350.96,100.30,6.00),vTravel,z5,tPen\WObj:=wPaper;
    MoveL Offs(pOrigin,350.96,100.30,0.00),v60,z0,tPen\WObj:=wPaper;
    MoveL Offs(pOrigin,345.40,105.86,0.00),v40,z0,tPen\WObj:=wPaper;
    MoveL Offs(pOrigin,345.72,105.57,0.00),v40,z0,tPen\WObj:=wPaper;
    MoveL Offs(pOrigin,353.23,113.09,0.00),v40,fine,tPen\WObj:=wPaper;
    MoveL Offs(pOrigin,353.23,113.09,6.00),v60,z5,tPen\WObj:=wPaper;
    MoveL Offs(pOrigin,352.85,114.22,6.00),vTravel,z5,tPen\WObj:=wPaper;
    MoveL Offs(pOrigin,352.85,114.22,0.00),v60,z0,tPen\WObj:=wPaper;
    MoveL Offs(pOrigin,353.06,114.65,0.00),v40,z0,tPen\WObj:=wPaper;
    MoveL Offs(pOrigin,352.85,114.22,0.00),v40,z0,tPen\WObj:=wPaper;
    MoveL Offs(pOrigin,353.27,114.86,0.00),v40,z0,tPen\WObj:=wPaper;
    MoveL Offs(pOrigin,353.49,115.29,0.00),v40,z0,tPen\WObj:=wPaper;
    MoveL Offs(pOrigin,353.27,114.86,0.00),v40,z0,tPen\WObj:=wPaper;
    MoveL Offs(pOrigin,353.49,115.29,0.00),v40,z0,tPen\WObj:=wPaper;
    MoveL Offs(pOrigin,353.70,116.35,0.00),v40,z0,tPen\WObj:=wPaper;
    MoveL Offs(pOrigin,354.12,116.56,0.00),v40,z0,tPen\WObj:=wPaper;
    MoveL Offs(pOrigin,354.12,116.56,0.00),v40,z0,tPen\WObj:=wPaper;
  ENDPROC

